C07287=1090.519,65.831,439.779,175.359,18.176,152.786
C07288=1090.524,66.080,439.762,175.361,18.177,152.786
C07289=1090.530,66.329,439.745,175.363,18.179,152.785
C07290=1090.536,66.579,439.729,175.365,18.181,152.785
C07291=1090.541,66.828,439.712,175.367,18.182,152.785
C07292=1090.547,67.078,439.696,175.369,18.183,152.785
C07293=1090.552,67.327,439.679,175.371,18.185,152.785
C07294=1090.559,67.576,439.662,175.373,18.187,152.785
C07295=1090.564,67.826,439.645,175.375,18.188,152.785
C07296=1090.570,68.075,439.629,175.377,18.189,152.785
C07297=1090.575,68.325,439.612,175.379,18.191,152.785
C07298=1090.581,68.574,439.596,175.381,18.192,152.785
C07299=1090.586,68.823,439.578,175.383,18.193,152.785
C07300=1090.592,69.072,439.562,175.385,18.195,152.785
C07301=1090.598,69.322,439.545,175.387,18.197,152.785
C07302=1090.604,69.571,439.528,175.389,18.198,152.785
C07303=1090.609,69.820,439.511,175.391,18.199,152.784
C07304=1090.615,70.070,439.495,175.393,18.201,152.784
C07305=1090.620,70.319,439.478,175.395,18.202,152.784
C07306=1090.627,70.568,439.461,175.397,18.204,152.784
C07307=1090.632,70.818,439.444,175.399,18.205,152.784
C07308=1090.638,71.067,439.428,175.401,18.207,152.784
C07309=1090.643,71.316,439.410,175.403,18.208,152.784
C07310=1090.648,71.566,439.394,175.405,18.210,152.784
C07311=1090.655,71.816,439.377,175.407,18.211,152.784
C07312=1090.660,72.065,439.359,175.409,18.213,152.784
C07313=1090.666,72.314,439.343,175.411,18.214,152.784
C07314=1090.672,72.564,439.326,175.413,18.216,152.784
C07315=1090.677,72.813,439.309,175.415,18.217,152.784
C07316=1090.683,73.062,439.292,175.417,18.218,152.783
C07317=1090.689,73.311,439.275,175.419,18.220,152.783
C07318=1090.694,73.561,439.258,175.421,18.222,152.783
C07319=1090.700,73.810,439.242,175.423,18.223,152.783
C07320=1090.705,74.059,439.224,175.425,18.224,152.783
C07321=1090.711,74.309,439.208,175.427,18.225,152.783
C07322=1090.717,74.559,439.190,175.430,18.227,152.783
C07323=1090.723,74.808,439.173,175.432,18.229,152.783
C07324=1090.729,75.057,439.156,175.433,18.230,152.783
C07325=1090.734,75.307,439.139,175.436,18.232,152.783
C07326=1090.740,75.556,439.122,175.438,18.233,152.783
C07327=1090.746,75.805,439.106,175.440,18.234,152.782
C07328=1090.751,76.054,439.088,175.442,18.236,152.782
C07329=1090.756,76.304,439.071,175.444,18.237,152.782
C07330=1090.762,76.553,439.053,175.446,18.239,152.782
C07331=1090.768,76.803,439.037,175.448,18.240,152.782
C07332=1090.774,77.052,439.019,175.450,18.241,152.782
C07333=1090.779,77.301,439.003,175.452,18.243,152.782
C07334=1090.785,77.550,438.986,175.454,18.244,152.782
C07335=1090.791,77.800,438.969,175.456,18.246,152.782
C07336=1090.797,78.050,438.951,175.458,18.247,152.782
C07337=1090.802,78.299,438.933,175.460,18.248,152.781
C07338=1090.808,78.548,438.917,175.462,18.249,152.781
C07339=1090.814,78.797,438.899,175.464,18.252,152.781
C07340=1090.819,79.047,438.883,175.466,18.253,152.781
C07341=1090.825,79.324,438.863,175.469,18.254,152.781
C07342=1090.832,79.600,438.844,175.471,18.256,152.781
C07343=1090.838,79.877,438.825,175.474,18.257,152.781
C07344=1090.845,80.153,438.805,175.476,18.259,152.781
C07345=1090.850,80.402,438.789,175.478,18.260,152.781
C07346=1090.855,80.651,438.771,175.480,18.262,152.781
C07347=1090.861,80.900,438.753,175.482,18.263,152.781
C07348=1090.867,81.151,438.736,175.484,18.265,152.781
C07349=1090.872,81.400,438.719,175.486,18.266,152.780
C07350=1090.878,81.649,438.701,175.488,18.268,152.780
C07351=1090.883,81.899,438.684,175.491,18.269,152.780
C07352=1090.888,82.148,438.667,175.492,18.270,152.780
C07353=1090.895,82.397,438.649,175.495,18.272,152.780
C07354=1090.901,82.647,438.633,175.496,18.273,152.780
C07355=1090.906,82.896,438.615,175.499,18.275,152.780
C07356=1090.912,83.145,438.597,175.501,18.276,152.780
C07357=1090.917,83.394,438.580,175.503,18.277,152.779
C07358=1090.923,83.644,438.563,175.505,18.278,152.779
C07359=1090.928,83.893,438.545,175.507,18.280,152.779
C07360=1090.934,84.142,438.527,175.510,18.282,152.779
C07361=1090.939,84.391,438.510,175.511,18.283,152.779
C07362=1090.946,84.641,438.492,175.514,18.284,152.779
C07363=1090.951,84.891,438.475,175.516,18.285,152.779
C07364=1090.956,85.140,438.458,175.518,18.287,152.779
C07365=1090.962,85.389,438.440,175.520,18.288,152.779
C07366=1090.968,85.639,438.422,175.522,18.290,152.778
C07367=1090.974,85.888,438.404,175.524,18.291,152.778
C07368=1090.980,86.136,438.388,175.526,18.292,152.778
C07369=1090.986,86.387,438.370,175.529,18.294,152.778
C07370=1090.991,86.636,438.353,175.530,18.295,152.778
C07371=1090.997,86.885,438.335,175.533,18.297,152.778
C07372=1091.002,87.134,438.318,175.535,18.298,152.778
C07373=1091.008,87.384,438.300,175.537,18.299,152.778
C07374=1091.014,87.633,438.282,175.539,18.300,152.778
C07375=1091.019,87.882,438.265,175.541,18.302,152.777
C07376=1091.025,88.131,438.247,175.543,18.303,152.777
C07377=1091.031,88.380,438.229,175.545,18.305,152.777
C07378=1091.036,88.629,438.211,175.548,18.306,152.777
C07379=1091.043,88.879,438.194,175.550,18.307,152.777
C07380=1091.048,89.129,438.177,175.552,18.309,152.777
C07381=1091.053,89.378,438.159,175.554,18.309,152.777
C07382=1091.059,89.628,438.141,175.556,18.311,152.777
C07383=1091.065,89.877,438.124,175.558,18.312,152.776
C07384=1091.070,90.126,438.106,175.561,18.314,152.776
C07385=1091.077,90.375,438.088,175.563,18.315,152.776
C07386=1091.082,90.624,438.071,175.565,18.316,152.776
C07387=1091.087,90.875,438.052,175.567,18.318,152.776
C07388=1091.093,91.124,438.034,175.569,18.319,152.776
C07389=1091.099,91.372,438.016,175.572,18.320,152.776
C07390=1091.105,91.622,437.998,175.573,18.321,152.775
C07391=1091.110,91.871,437.981,175.576,18.323,152.775
C07392=1091.116,92.120,437.963,175.578,18.324,152.775
C07393=1091.121,92.370,437.945,175.580,18.326,152.775
C07394=1091.127,92.619,437.927,175.582,18.327,152.775
C07395=1091.132,92.868,437.909,175.584,18.328,152.775
C07396=1091.139,93.118,437.891,175.587,18.330,152.775
C07397=1091.144,93.367,437.874,175.589,18.331,152.775
C07398=1091.149,93.616,437.856,175.591,18.332,152.774
C07399=1091.155,93.866,437.838,175.593,18.334,152.774
C07400=1091.161,94.114,437.820,175.595,18.335,152.774
C07401=1091.167,94.364,437.802,175.598,18.336,152.774
C07402=1091.172,94.613,437.783,175.599,18.337,152.774
C07403=1091.177,94.862,437.766,175.602,18.339,152.774
C07404=1091.183,95.112,437.748,175.604,18.341,152.774
C07405=1091.189,95.389,437.727,175.607,18.342,152.773
C07406=1091.196,95.666,437.708,175.609,18.343,152.773
C07407=1091.202,95.942,437.688,175.611,18.344,152.773
C07408=1091.208,96.219,437.667,175.614,18.346,152.773
C07409=1091.214,96.468,437.650,175.616,18.347,152.773
C07410=1091.220,96.717,437.632,175.618,18.348,152.773
C07411=1091.225,96.966,437.614,175.621,18.350,152.773
C07412=1091.230,97.215,437.595,175.623,18.351,152.772
C07413=1091.236,97.465,437.577,175.625,18.352,152.772
C07414=1091.242,97.714,437.560,175.627,18.354,152.772
C07415=1091.247,97.964,437.541,175.629,18.355,152.772
C07416=1091.253,98.212,437.523,175.632,18.356,152.772
C07417=1091.259,98.462,437.505,175.634,18.358,152.772
C07418=1091.265,98.711,437.488,175.636,18.358,152.772
C07419=1091.271,98.961,437.468,175.638,18.360,152.771
C07420=1091.276,99.210,437.451,175.640,18.361,152.771
C07421=1091.282,99.459,437.433,175.643,18.362,152.771
C07422=1091.287,99.708,437.414,175.645,18.364,152.771
C07423=1091.293,99.958,437.396,175.647,18.365,152.771
C07424=1091.299,100.207,437.378,175.649,18.367,152.771
C07425=1091.305,100.456,437.359,175.651,18.367,152.770
C07426=1091.310,100.705,437.342,175.654,18.369,152.770
C07427=1091.316,100.955,437.324,175.656,18.370,152.770
C07428=1091.321,101.204,437.305,175.658,18.371,152.770
C07429=1091.327,101.454,437.287,175.661,18.373,152.770
C07430=1091.333,101.702,437.268,175.662,18.374,152.770
C07431=1091.339,101.952,437.250,175.665,18.375,152.769
C07432=1091.343,102.201,437.232,175.668,18.376,152.769
C07433=1091.350,102.451,437.213,175.669,18.377,152.769
C07434=1091.355,102.700,437.195,175.672,18.379,152.769
C07435=1091.361,102.949,437.176,175.675,18.380,152.769
C07436=1091.366,103.198,437.158,175.676,18.381,152.769
C07437=1091.372,103.448,437.140,175.679,18.383,152.769
C07438=1091.377,103.697,437.121,175.681,18.383,152.768
C07439=1091.383,103.946,437.103,175.683,18.385,152.768
C07440=1091.388,104.195,437.085,175.686,18.387,152.768
C07441=1091.395,104.444,437.066,175.688,18.387,152.768
C07442=1091.399,104.694,437.048,175.690,18.389,152.768
C07443=1091.406,104.943,437.029,175.693,18.390,152.768
C07444=1091.411,105.192,437.011,175.694,18.391,152.767
C07445=1091.417,105.441,436.992,175.697,18.393,152.767
C07446=1091.422,105.691,436.974,175.699,18.393,152.767
C07447=1091.428,105.940,436.956,175.701,18.395,152.767
C07448=1091.433,106.189,436.937,175.704,18.396,152.767
C07449=1091.439,106.439,436.918,175.706,18.397,152.767
C07450=1091.445,106.688,436.900,175.708,18.399,152.766
C07451=1091.450,106.937,436.881,175.711,18.400,152.766
C07452=1091.456,107.186,436.863,175.713,18.401,152.766
C07453=1091.461,107.435,436.844,175.715,18.402,152.766
C07454=1091.468,107.685,436.826,175.718,18.404,152.766
C07455=1091.473,107.934,436.807,175.720,18.405,152.766
C07456=1091.478,108.183,436.788,175.722,18.406,152.765
C07457=1091.484,108.433,436.770,175.724,18.407,152.765
C07458=1091.490,108.681,436.751,175.727,18.408,152.765
C07459=1091.496,108.931,436.732,175.729,18.410,152.765
C07460=1091.501,109.181,436.714,175.731,18.410,152.765
C07461=1091.506,109.429,436.695,175.734,18.412,152.764
C07462=1091.513,109.678,436.676,175.736,18.413,152.764
C07463=1091.518,109.928,436.658,175.738,18.414,152.764
C07464=1091.524,110.177,436.639,175.741,18.415,152.764
C07465=1091.530,110.426,436.620,175.743,18.417,152.764
C07466=1091.535,110.675,436.601,175.745,18.417,152.763
C07467=1091.541,110.925,436.583,175.748,18.419,152.763
C07468=1091.547,111.174,436.564,175.750,18.420,152.763
C07469=1091.553,111.451,436.544,175.752,18.421,152.763
C07470=1091.560,111.727,436.522,175.755,18.422,152.763
C07471=1091.566,112.004,436.502,175.757,18.424,152.763
C07472=1091.572,112.281,436.481,175.760,18.425,152.762
C07473=1091.578,112.530,436.462,175.763,18.426,152.762
C07474=1091.583,112.779,436.443,175.765,18.428,152.762
C07475=1091.588,113.029,436.425,175.767,18.428,152.762
C07476=1091.595,113.278,436.406,175.770,18.430,152.762
C07477=1091.600,113.527,436.387,175.772,18.431,152.761
C07478=1091.605,113.776,436.368,175.774,18.432,152.761
C07479=1091.611,114.025,436.349,175.777,18.433,152.761
C07480=1091.617,114.275,436.330,175.779,18.435,152.761
C07481=1091.623,114.523,436.311,175.781,18.435,152.761
C07482=1091.628,114.773,436.292,175.784,18.437,152.760
C07483=1091.634,115.023,436.273,175.786,18.438,152.760
C07484=1091.639,115.272,436.254,175.788,18.439,152.760
C07485=1091.644,115.521,436.235,175.791,18.440,152.760
C07486=1091.650,115.770,436.216,175.793,18.442,152.760
C07487=1091.655,116.019,436.197,175.795,18.442,152.759
C07488=1091.661,116.269,436.178,175.798,18.444,152.759
C07489=1091.667,116.518,436.158,175.801,18.445,152.759
C07490=1091.672,116.767,436.140,175.802,18.446,152.759
C07491=1091.677,117.016,436.120,175.805,18.447,152.759
C07492=1091.684,117.265,436.102,175.808,18.448,152.758
C07493=1091.689,117.514,436.083,175.809,18.450,152.758
C07494=1091.694,117.763,436.064,175.812,18.451,152.758
C07495=1091.700,118.013,436.044,175.815,18.452,152.758
C07496=1091.705,118.262,436.025,175.816,18.453,152.758
C07497=1091.711,118.511,436.006,175.819,18.454,152.757
C07498=1091.717,118.760,435.987,175.822,18.456,152.757
C07499=1091.722,119.010,435.968,175.824,18.456,152.757
C07500=1091.727,119.259,435.949,175.826,18.458,152.757
C07501=1091.733,119.508,435.930,175.829,18.459,152.757
C07502=1091.739,119.758,435.910,175.832,18.460,152.756
C07503=1091.744,120.007,435.891,175.833,18.461,152.756
C07504=1091.750,120.256,435.872,175.836,18.462,152.756
C07505=1091.756,120.504,435.852,175.839,18.463,152.756
C07506=1091.761,120.754,435.833,175.840,18.464,152.756
C07507=1091.767,121.003,435.814,175.843,18.465,152.755
C07508=1091.772,121.252,435.795,175.846,18.467,152.755
C07509=1091.778,121.502,435.776,175.848,18.468,152.755
C07510=1091.783,121.751,435.756,175.850,18.469,152.755
C07511=1091.789,122.000,435.737,175.853,18.470,152.755
C07512=1091.795,122.249,435.717,175.855,18.471,152.754
C07513=1091.800,122.498,435.698,175.858,18.472,152.754
C07514=1091.806,122.747,435.679,175.860,18.473,152.754
C07515=1091.812,122.997,435.660,175.863,18.474,152.754
C07516=1091.817,123.246,435.641,175.865,18.475,152.754
C07517=1091.823,123.495,435.621,175.867,18.477,152.753
C07518=1091.828,123.744,435.601,175.870,18.478,152.753
C07519=1091.833,123.994,435.582,175.872,18.478,152.753
C07520=1091.839,124.243,435.563,175.875,18.480,152.753
C07521=1091.845,124.492,435.543,175.877,18.481,152.752
C07522=1091.851,124.741,435.524,175.879,18.482,152.752
C07523=1091.856,124.991,435.504,175.882,18.483,152.752
C07524=1091.862,125.239,435.484,175.885,18.484,152.752
C07525=1091.867,125.488,435.465,175.887,18.485,152.751
C07526=1091.873,125.738,435.446,175.889,18.486,152.751
C07527=1091.879,125.986,435.426,175.892,18.487,152.751
C07528=1091.885,126.236,435.407,175.895,18.488,152.751
C07529=1091.890,126.485,435.388,175.897,18.489,152.750
C07530=1091.896,126.734,435.367,175.899,18.490,152.750
C07531=1091.901,126.984,435.348,175.902,18.492,152.750
C07532=1091.907,127.233,435.329,175.904,18.492,152.750
C07533=1091.913,127.509,435.308,175.907,18.494,152.750
C07534=1091.920,127.786,435.285,175.910,18.495,152.749
C07535=1091.926,128.063,435.263,175.913,18.496,152.749
C07536=1091.932,128.339,435.242,175.916,18.497,152.749
C07537=1091.938,128.588,435.223,175.917,18.498,152.749
C07538=1091.943,128.838,435.202,175.920,18.499,152.748
C07539=1091.949,129.087,435.183,175.923,18.500,152.748
C07540=1091.955,129.336,435.163,175.925,18.501,152.748
C07541=1091.961,129.585,435.144,175.928,18.502,152.747
C07542=1091.967,129.834,435.124,175.930,18.503,152.747
C07543=1091.972,130.084,435.105,175.933,18.504,152.747
C07544=1091.978,130.332,435.085,175.935,18.505,152.747
C07545=1091.983,130.582,435.065,175.938,18.506,152.746
C07546=1091.989,130.831,435.045,175.940,18.507,152.746
C07547=1091.995,131.080,435.026,175.942,18.508,152.746
C07548=1092.001,131.329,435.006,175.945,18.509,152.746
C07549=1092.007,131.579,434.986,175.948,18.510,152.746
C07550=1092.012,131.828,434.966,175.950,18.511,152.745
C07551=1092.018,132.077,434.947,175.952,18.512,152.745
C07552=1092.024,132.326,434.927,175.955,18.513,152.745
C07553=1092.029,132.575,434.907,175.958,18.514,152.744
C07554=1092.035,132.824,434.887,175.961,18.515,152.744
C07555=1092.041,133.073,434.867,175.962,18.516,152.744
C07556=1092.046,133.323,434.848,175.965,18.517,152.744
C07557=1092.052,133.572,434.827,175.968,18.518,152.743
C07558=1092.057,133.821,434.808,175.971,18.519,152.743
C07559=1092.062,134.070,434.787,175.973,18.520,152.743
C07560=1092.068,134.319,434.767,175.975,18.521,152.743
C07561=1092.074,134.569,434.748,175.978,18.522,152.742
C07562=1092.079,134.818,434.727,175.981,18.523,152.742
C07563=1092.085,135.067,434.708,175.983,18.524,152.742
C07564=1092.090,135.316,434.688,175.986,18.525,152.742
C07565=1092.096,135.565,434.668,175.988,18.526,152.741
C07566=1092.102,135.814,434.648,175.991,18.527,152.741
C07567=1092.108,136.063,434.627,175.993,18.528,152.741
C07568=1092.113,136.313,434.608,175.996,18.529,152.741
C07569=1092.119,136.562,434.587,175.998,18.530,152.740
C07570=1092.125,136.810,434.567,176.001,18.531,152.740
C07571=1092.131,137.059,434.547,176.003,18.532,152.740
C07572=1092.135,137.309,434.528,176.006,18.533,152.740
C07573=1092.141,137.558,434.508,176.009,18.534,152.739
C07574=1092.147,137.807,434.487,176.011,18.535,152.739
C07575=1092.153,138.056,434.467,176.013,18.536,152.739
C07576=1092.158,138.306,434.447,176.016,18.537,152.739
C07577=1092.164,138.554,434.427,176.019,18.538,152.738
C07578=1092.169,138.803,434.407,176.021,18.539,152.738
C07579=1092.175,139.052,434.387,176.024,18.539,152.738
C07580=1092.180,139.301,434.366,176.026,18.540,152.737
C07581=1092.187,139.551,434.346,176.029,18.541,152.737
C07582=1092.192,139.801,434.326,176.032,18.543,152.737
C07583=1092.198,140.049,434.306,176.034,18.543,152.737
C07584=1092.203,140.299,434.286,176.037,18.544,152.736
C07585=1092.209,140.547,434.266,176.039,18.545,152.736
C07586=1092.214,140.797,434.245,176.042,18.547,152.736
C07587=1092.219,141.046,434.225,176.045,18.548,152.736
C07588=1092.225,141.294,434.205,176.047,18.548,152.735
C07589=1092.231,141.544,434.184,176.050,18.549,152.735
C07590=1092.237,141.792,434.164,176.052,18.550,152.735
C07591=1092.242,142.042,434.144,176.055,18.551,152.734
C07592=1092.248,142.291,434.123,176.057,18.552,152.734
C07593=1092.254,142.540,434.103,176.060,18.553,152.734
C07594=1092.259,142.789,434.082,176.063,18.554,152.734
C07595=1092.264,143.038,434.062,176.065,18.555,152.733
C07596=1092.270,143.287,434.042,176.068,18.556,152.733
C07597=1092.276,143.564,434.019,176.071,18.557,152.733
C07598=1092.282,143.841,433.996,176.074,18.558,152.732
C07599=1092.289,144.118,433.974,176.077,18.559,152.732
C07600=1092.295,144.394,433.951,176.080,18.560,152.732
C07601=1092.301,144.643,433.930,176.082,18.561,152.731
C07602=1092.306,144.892,433.910,176.085,18.562,152.731
C07603=1092.312,145.141,433.890,176.087,18.563,152.731
C07604=1092.317,145.390,433.869,176.090,18.564,152.731
C07605=1092.322,145.639,433.849,176.093,18.564,152.730
C07606=1092.329,145.889,433.828,176.095,18.566,152.730
C07607=1092.334,146.137,433.807,176.097,18.566,152.730
C07608=1092.340,146.387,433.787,176.100,18.567,152.730
C07609=1092.346,146.635,433.767,176.103,18.568,152.729
C07610=1092.351,146.884,433.746,176.106,18.569,152.729
C07611=1092.357,147.134,433.725,176.109,18.570,152.729
C07612=1092.362,147.383,433.705,176.111,18.571,152.728
C07613=1092.368,147.632,433.684,176.114,18.571,152.728
C07614=1092.374,147.881,433.663,176.116,18.573,152.728
C07615=1092.379,148.130,433.643,176.119,18.574,152.727
C07616=1092.385,148.380,433.622,176.122,18.574,152.727
C07617=1092.391,148.628,433.602,176.125,18.575,152.727
C07618=1092.396,148.877,433.581,176.127,18.576,152.727
C07619=1092.402,149.126,433.560,176.129,18.577,152.726
C07620=1092.407,149.376,433.539,176.132,18.578,152.726
C07621=1092.413,149.625,433.519,176.135,18.579,152.726
C07622=1092.418,149.874,433.497,176.138,18.580,152.725
C07623=1092.424,150.122,433.477,176.140,18.581,152.725
C07624=1092.430,150.372,433.457,176.143,18.581,152.725
C07625=1092.435,150.621,433.436,176.146,18.582,152.724
C07626=1092.441,150.870,433.415,176.148,18.584,152.724
C07627=1092.446,151.119,433.394,176.151,18.584,152.724
C07628=1092.452,151.369,433.373,176.153,18.585,152.724
C07629=1092.458,151.617,433.352,176.156,18.586,152.723
C07630=1092.463,151.866,433.331,176.159,18.587,152.723
C07631=1092.468,152.116,433.311,176.162,18.588,152.723
C07632=1092.474,152.365,433.289,176.164,18.589,152.722
C07633=1092.479,152.614,433.269,176.167,18.590,152.722
C07634=1092.486,152.862,433.248,176.169,18.590,152.722
C07635=1092.491,153.111,433.227,176.172,18.591,152.721
C07636=1092.497,153.361,433.206,176.175,18.592,152.721
C07637=1092.502,153.610,433.185,176.178,18.593,152.721
C07638=1092.508,153.859,433.165,176.181,18.594,152.720
C07639=1092.514,154.108,433.143,176.184,18.595,152.720
C07640=1092.519,154.357,433.122,176.186,18.595,152.720
C07641=1092.525,154.605,433.101,176.189,18.596,152.719
C07642=1092.531,154.855,433.080,176.191,18.597,152.719
C07643=1092.536,155.104,433.059,176.194,18.598,152.719
C07644=1092.541,155.353,433.038,176.197,18.599,152.719
C07645=1092.548,155.602,433.017,176.200,18.600,152.718
C07646=1092.553,155.851,432.996,176.202,18.600,152.718
C07647=1092.558,156.100,432.975,176.205,18.601,152.718
C07648=1092.564,156.350,432.954,176.208,18.602,152.717
C07649=1092.570,156.598,432.933,176.210,18.603,152.717
C07650=1092.575,156.847,432.912,176.213,18.604,152.717
C07651=1092.581,157.096,432.891,176.216,18.605,152.716
C07652=1092.586,157.346,432.869,176.219,18.606,152.716
C07653=1092.591,157.594,432.848,176.221,18.606,152.716
C07654=1092.597,157.844,432.827,176.224,18.607,152.715
C07655=1092.603,158.093,432.806,176.227,18.608,152.715
C07656=1092.608,158.341,432.785,176.230,18.609,152.715
C07657=1092.614,158.591,432.764,176.233,18.610,152.714
C07658=1092.620,158.840,432.743,176.235,18.611,152.714
C07659=1092.626,159.089,432.721,176.237,18.612,152.714
C07660=1092.631,159.338,432.700,176.240,18.612,152.713
C07661=1092.637,159.614,432.676,176.244,18.613,152.713
C07662=1092.643,159.891,432.653,176.247,18.615,152.713
C07663=1092.650,160.167,432.630,176.250,18.615,152.712
C07664=1092.656,160.443,432.606,176.253,18.616,152.712
C07665=1092.662,160.692,432.584,176.256,18.617,152.712
C07666=1092.667,160.941,432.563,176.259,18.618,152.711
C07667=1092.673,161.191,432.541,176.261,18.619,152.711
C07668=1092.678,161.439,432.520,176.263,18.619,152.711
C07669=1092.684,161.688,432.499,176.266,18.620,152.710
C07670=1092.690,161.938,432.478,176.269,18.621,152.710
C07671=1092.694,162.186,432.456,176.272,18.622,152.710
C07672=1092.700,162.435,432.435,176.275,18.622,152.709
C07673=1092.706,162.684,432.413,176.278,18.624,152.709
C07674=1092.711,162.933,432.392,176.281,18.624,152.709
C07675=1092.717,163.183,432.370,176.283,18.625,152.708
C07676=1092.722,163.432,432.348,176.286,18.627,152.708
C07677=1092.727,163.680,432.327,176.288,18.627,152.708
C07678=1092.733,163.929,432.305,176.291,18.628,152.707
C07679=1092.738,164.178,432.284,176.294,18.628,152.707
C07680=1092.744,164.428,432.263,176.297,18.630,152.707
C07681=1092.749,164.677,432.241,176.300,18.630,152.706
C07682=1092.754,164.925,432.220,176.303,18.631,152.706
C07683=1092.760,165.175,432.197,176.306,18.632,152.706
C07684=1092.765,165.423,432.176,176.308,18.633,152.705
C07685=1092.772,165.672,432.154,176.311,18.634,152.705
C07686=1092.776,165.921,432.133,176.313,18.634,152.705
C07687=1092.783,166.170,432.111,176.316,18.635,152.704
C07688=1092.787,166.419,432.089,176.319,18.636,152.704
C07689=1092.794,166.668,432.067,176.322,18.637,152.704
C07690=1092.798,166.917,432.046,176.325,18.638,152.703
C07691=1092.804,167.166,432.024,176.328,18.639,152.703
C07692=1092.809,167.415,432.002,176.331,18.639,152.703
C07693=1092.815,167.664,431.981,176.333,18.641,152.702
C07694=1092.820,167.913,431.959,176.336,18.641,152.702
C07695=1092.826,168.162,431.937,176.339,18.642,152.702
C07696=1092.831,168.411,431.915,176.341,18.642,152.701
C07697=1092.837,168.660,431.894,176.344,18.643,152.701
C07698=1092.842,168.909,431.872,176.347,18.644,152.701
C07699=1092.848,169.158,431.850,176.350,18.645,152.700
C07700=1092.853,169.407,431.828,176.353,18.646,152.700
C07701=1092.859,169.657,431.806,176.356,18.647,152.700
C07702=1092.864,169.905,431.785,176.359,18.647,152.699
C07703=1092.870,170.155,431.763,176.362,18.648,152.699
C07704=1092.875,170.403,431.741,176.365,18.649,152.699
C07705=1092.881,170.653,431.719,176.368,18.650,152.698
C07706=1092.887,170.901,431.697,176.371,18.651,152.698
C07707=1092.893,171.150,431.675,176.373,18.652,152.697
C07708=1092.898,171.399,431.653,176.375,18.652,152.697
C07709=1092.904,171.648,431.632,176.378,18.652,152.697
C07710=1092.909,171.898,431.609,176.381,18.654,152.696
C07711=1092.915,172.146,431.588,176.384,18.654,152.696
C07712=1092.920,172.395,431.565,176.387,18.655,152.696
C07713=1092.926,172.643,431.544,176.390,18.656,152.695
C07714=1092.931,172.893,431.522,176.393,18.657,152.695
C07715=1092.937,173.142,431.500,176.396,18.657,152.695
C07716=1092.943,173.390,431.478,176.399,18.658,152.694
C07717=1092.948,173.640,431.455,176.402,18.659,152.694
C07718=1092.954,173.888,431.434,176.405,18.660,152.693
C07719=1092.959,174.138,431.412,176.408,18.661,152.693
C07720=1092.965,174.387,431.389,176.411,18.661,152.693
C07721=1092.970,174.635,431.368,176.413,18.662,152.692
C07722=1092.976,174.885,431.345,176.416,18.662,152.692
C07723=1092.982,175.133,431.323,176.419,18.663,152.692
C07724=1092.987,175.382,431.301,176.422,18.664,152.691
C07725=1092.994,175.659,431.277,176.425,18.665,152.691
C07726=1093.000,175.934,431.252,176.428,18.666,152.690
C07727=1093.006,176.210,431.227,176.431,18.666,152.690
C07728=1093.013,176.486,431.203,176.434,18.667,152.690
C07729=1093.018,176.735,431.180,176.437,18.668,152.689
C07730=1093.023,176.984,431.158,176.440,18.668,152.689
C07731=1093.029,177.233,431.137,176.443,18.669,152.689
C07732=1093.035,177.482,431.114,176.446,18.670,152.688
C07733=1093.040,177.732,431.092,176.449,18.671,152.688
C07734=1093.046,177.980,431.070,176.452,18.671,152.687
C07735=1093.052,178.229,431.047,176.455,18.672,152.687
C07736=1093.057,178.478,431.025,176.458,18.673,152.687
C07737=1093.064,178.727,431.003,176.461,18.673,152.686
C07738=1093.069,178.975,430.980,176.464,18.674,152.686
C07739=1093.074,179.225,430.958,176.467,18.675,152.685
C07740=1093.081,179.473,430.936,176.470,18.676,152.685
C07741=1093.086,179.723,430.913,176.473,18.677,152.685
C07742=1093.091,179.971,430.891,176.476,18.677,152.684
C07743=1093.097,180.220,430.869,176.479,18.678,152.684
C07744=1093.103,180.469,430.846,176.482,18.679,152.683
C07745=1093.109,180.719,430.824,176.485,18.679,152.683
C07746=1093.114,180.968,430.801,176.488,18.680,152.683
C07747=1093.120,181.216,430.779,176.490,18.680,152.682
C07748=1093.126,181.465,430.757,176.493,18.681,152.682
C07749=1093.131,181.714,430.734,176.496,18.681,152.681
C07750=1093.137,181.964,430.712,176.499,18.682,152.681
C07751=1093.143,182.212,430.689,176.502,18.683,152.681
C07752=1093.149,182.461,430.666,176.505,18.683,152.680
C07753=1093.154,182.710,430.645,176.508,18.684,152.680
C07754=1093.159,182.959,430.622,176.511,18.685,152.679
C07755=1093.166,183.207,430.599,176.514,18.685,152.679
C07756=1093.171,183.457,430.577,176.517,18.686,152.679
C07757=1093.177,183.706,430.554,176.520,18.687,152.678
C07758=1093.183,183.955,430.531,176.523,18.688,152.678
C07759=1093.189,184.203,430.509,176.526,18.688,152.677
C07760=1093.194,184.452,430.487,176.529,18.689,152.677
C07761=1093.200,184.701,430.464,176.532,18.690,152.677
C07762=1093.206,184.950,430.441,176.535,18.690,152.676
C07763=1093.211,185.199,430.418,176.538,18.691,152.676
C07764=1093.217,185.448,430.396,176.541,18.692,152.675
C07765=1093.222,185.697,430.373,176.544,18.692,152.675
C07766=1093.228,185.945,430.350,176.547,18.693,152.675
C07767=1093.233,186.194,430.327,176.550,18.694,152.674
C07768=1093.239,186.443,430.304,176.553,18.694,152.674
C07769=1093.244,186.693,430.282,176.556,18.695,152.673
C07770=1093.250,186.942,430.259,176.559,18.696,152.673
C07771=1093.255,187.190,430.237,176.562,18.697,152.673
C07772=1093.261,187.439,430.214,176.565,18.697,152.672
C07773=1093.266,187.688,430.190,176.568,18.698,152.672
C07774=1093.272,187.937,430.167,176.571,18.699,152.672
C07775=1093.277,188.186,430.145,176.574,18.699,152.671
C07776=1093.283,188.435,430.122,176.577,18.700,152.671
C07777=1093.288,188.683,430.100,176.580,18.701,152.670
C07778=1093.294,188.932,430.077,176.583,18.701,152.670
C07779=1093.300,189.181,430.054,176.586,18.702,152.670
C07780=1093.305,189.430,430.030,176.589,18.703,152.669
C07781=1093.310,189.679,430.007,176.592,18.704,152.669
C07782=1093.316,189.928,429.984,176.595,18.704,152.668
C07783=1093.322,190.177,429.961,176.598,18.705,152.668
C07784=1093.327,190.425,429.939,176.601,18.706,152.668
C07785=1093.333,190.674,429.916,176.604,18.706,152.667
C07786=1093.338,190.923,429.892,176.607,18.707,152.667
C07787=1093.343,191.172,429.869,176.610,18.708,152.666
C07788=1093.349,191.421,429.846,176.613,18.709,152.666
C07789=1093.355,191.697,429.821,176.616,18.709,152.666
C07790=1093.361,191.972,429.796,176.619,18.710,152.665
C07791=1093.368,192.248,429.769,176.623,18.711,152.665
C07792=1093.374,192.524,429.744,176.626,18.712,152.664
C07793=1093.379,192.773,429.721,176.629,18.712,152.664
C07794=1093.385,193.021,429.698,176.632,18.713,152.663
C07795=1093.391,193.270,429.675,176.635,18.714,152.663
C07796=1093.396,193.520,429.651,176.638,18.714,152.663
C07797=1093.402,193.768,429.628,176.641,18.715,152.662
C07798=1093.407,194.017,429.605,176.644,18.716,152.662
C07799=1093.413,194.266,429.582,176.647,18.716,152.661
C07800=1093.418,194.515,429.558,176.650,18.717,152.661
C07801=1093.424,194.764,429.535,176.653,18.718,152.661
C07802=1093.430,195.013,429.512,176.656,18.718,152.660
C07803=1093.436,195.261,429.489,176.660,18.719,152.660
C07804=1093.441,195.510,429.465,176.663,18.719,152.659
C07805=1093.446,195.759,429.442,176.666,18.721,152.659
C07806=1093.452,196.008,429.419,176.669,18.721,152.658
C07807=1093.458,196.256,429.396,176.672,18.722,152.658
C07808=1093.463,196.505,429.372,176.675,18.723,152.658
C07809=1093.469,196.754,429.349,176.678,18.723,152.657
C07810=1093.475,197.003,429.326,176.681,18.724,152.657
C07811=1093.480,197.252,429.302,176.685,18.724,152.656
C07812=1093.486,197.501,429.279,176.688,18.725,152.656
C07813=1093.491,197.750,429.256,176.691,18.726,152.655
C07814=1093.497,197.998,429.232,176.694,18.726,152.655
C07815=1093.502,198.247,429.209,176.697,18.727,152.655
C07816=1093.508,198.496,429.186,176.700,18.728,152.654
C07817=1093.514,198.744,429.162,176.703,18.728,152.654
C07818=1093.519,198.993,429.139,176.706,18.728,152.653
C07819=1093.526,199.242,429.115,176.709,18.729,152.653
C07820=1093.531,199.492,429.091,176.713,18.730,152.653
C07821=1093.537,199.741,429.068,176.716,18.731,152.652
C07822=1093.543,199.989,429.045,176.719,18.731,152.652
C07823=1093.548,200.238,429.021,176.722,18.732,152.651
C07824=1093.554,200.486,428.997,176.725,18.733,152.651
C07825=1093.559,200.735,428.974,176.728,18.733,152.650
C07826=1093.565,200.984,428.950,176.731,18.734,152.650
C07827=1093.571,201.233,428.927,176.734,18.734,152.649
C07828=1093.577,201.482,428.903,176.737,18.735,152.649
C07829=1093.582,201.731,428.880,176.740,18.736,152.649
C07830=1093.588,201.979,428.856,176.743,18.736,152.648
C07831=1093.593,202.228,428.832,176.746,18.737,152.648
C07832=1093.599,202.477,428.809,176.749,18.737,152.647
C07833=1093.605,202.726,428.786,176.753,18.738,152.647
C07834=1093.611,202.975,428.761,176.756,18.739,152.646
C07835=1093.616,203.224,428.738,176.759,18.739,152.646
C07836=1093.622,203.472,428.714,176.762,18.740,152.646
C07837=1093.627,203.721,428.690,176.765,18.741,152.645
C07838=1093.633,203.970,428.667,176.768,18.741,152.645
C07839=1093.638,204.218,428.643,176.772,18.742,152.644
C07840=1093.644,204.468,428.619,176.775,18.742,152.644
C07841=1093.650,204.717,428.595,176.778,18.743,152.643
C07842=1093.655,204.965,428.571,176.781,18.744,152.643
C07843=1093.661,205.214,428.548,176.784,18.745,152.643
C07844=1093.666,205.463,428.524,176.788,18.745,152.642
C07845=1093.671,205.711,428.499,176.791,18.746,152.642
C07846=1093.678,205.961,428.476,176.794,18.747,152.641
C07847=1093.683,206.209,428.452,176.797,18.747,152.641
C07848=1093.689,206.458,428.428,176.800,18.748,152.641
C07849=1093.694,206.706,428.404,176.803,18.748,152.640
C07850=1093.699,206.955,428.380,176.806,18.749,152.640
C07851=1093.706,207.204,428.356,176.810,18.750,152.639
C07852=1093.711,207.453,428.332,176.813,18.751,152.639
C07853=1093.734,208.471,428.234,176.870,18.776,152.634
C07854=1093.742,208.846,428.197,176.874,18.778,152.634
C07855=1093.751,209.221,428.161,176.878,18.781,152.633
C07856=1093.759,209.597,428.124,176.884,18.784,152.633
C07857=1093.768,209.972,428.087,176.888,18.785,152.633
C07858=1093.773,210.221,428.063,176.891,18.787,152.632
C07859=1093.779,210.470,428.038,176.894,18.789,152.632
C07860=1093.785,210.719,428.014,176.897,18.790,152.632
C07861=1093.791,210.968,427.989,176.899,18.791,152.632
C07862=1093.796,211.217,427.965,176.903,18.793,152.632
C07863=1093.801,211.465,427.941,176.906,18.794,152.631
C07864=1093.807,211.714,427.916,176.909,18.796,152.631
C07865=1093.813,211.962,427.891,176.912,18.798,152.631
C07866=1093.818,212.211,427.867,176.915,18.799,152.631
C07867=1093.824,212.460,427.842,176.918,18.801,152.630
C07868=1093.829,212.709,427.818,176.921,18.802,152.630
C07869=1093.835,212.958,427.793,176.924,18.804,152.630
C07870=1093.841,213.206,427.768,176.927,18.805,152.630
C07871=1093.847,213.455,427.744,176.930,18.807,152.630
C07872=1093.852,213.704,427.720,176.933,18.808,152.629
C07873=1093.857,213.953,427.695,176.936,18.810,152.629
C07874=1093.863,214.202,427.671,176.939,18.811,152.629
C07875=1093.869,214.450,427.646,176.942,18.813,152.629
C07876=1093.875,214.699,427.621,176.945,18.815,152.629
C07877=1093.880,214.948,427.597,176.948,18.816,152.628
C07878=1093.886,215.196,427.572,176.951,18.818,152.628
C07879=1093.891,215.445,427.547,176.954,18.819,152.628
C07880=1093.897,215.694,427.523,176.958,18.821,152.628
C07881=1093.902,215.943,427.497,176.960,18.823,152.628
C07882=1093.907,216.191,427.473,176.964,18.824,152.627
C07883=1093.913,216.440,427.448,176.966,18.825,152.627
C07884=1093.919,216.688,427.423,176.969,18.827,152.627
C07885=1093.925,216.938,427.399,176.972,18.829,152.627
C07886=1093.930,217.186,427.374,176.975,18.830,152.627
C07887=1093.936,217.435,427.348,176.978,18.832,152.626
C07888=1093.941,217.684,427.324,176.981,18.833,152.626
C07889=1093.947,217.933,427.299,176.985,18.835,152.626
C07890=1093.952,218.181,427.275,176.987,18.837,152.626
C07891=1093.959,218.430,427.249,176.991,18.838,152.626
C07892=1093.964,218.678,427.225,176.994,18.840,152.625
C07893=1093.969,218.927,427.199,176.997,18.841,152.625
C07894=1093.975,219.176,427.175,177.000,18.843,152.625
C07895=1093.981,219.425,427.149,177.003,18.845,152.625
C07896=1093.986,219.673,427.125,177.006,18.846,152.624
C07897=1093.992,219.922,427.100,177.009,18.848,152.624
C07898=1093.997,220.170,427.074,177.012,18.849,152.624
C07899=1094.003,220.419,427.050,177.015,18.850,152.624
C07900=1094.009,220.667,427.025,177.018,18.852,152.624
C07901=1094.015,220.917,427.000,177.021,18.854,152.623
C07902=1094.020,221.166,426.974,177.024,18.855,152.623
C07903=1094.026,221.414,426.949,177.027,18.857,152.623
C07904=1094.032,221.663,426.925,177.030,18.859,152.623
C07905=1094.037,221.911,426.900,177.033,18.860,152.623
C07906=1094.046,222.291,426.861,177.038,18.863,152.622
C07907=1094.054,222.670,426.822,177.043,18.865,152.622
C07908=1094.063,223.049,426.784,177.047,18.867,152.622
C07909=1094.072,223.430,426.745,177.052,18.870,152.621
C07910=1094.077,223.678,426.720,177.055,18.871,152.621
C07911=1094.082,223.927,426.695,177.058,18.873,152.621
C07912=1094.088,224.175,426.670,177.061,18.875,152.621
C07913=1094.093,224.424,426.644,177.064,18.877,152.621
C07914=1094.100,224.673,426.619,177.067,18.878,152.620
C07915=1094.104,224.922,426.594,177.071,18.880,152.620
C07916=1094.110,225.170,426.569,177.073,18.881,152.620
C07917=1094.117,225.419,426.543,177.077,18.883,152.620
C07918=1094.121,225.667,426.518,177.079,18.884,152.620
C07919=1094.128,225.916,426.492,177.083,18.886,152.619
C07920=1094.132,226.164,426.467,177.085,18.888,152.619
C07921=1094.138,226.413,426.442,177.089,18.889,152.619
C07922=1094.144,226.662,426.416,177.092,18.891,152.619
C07923=1094.150,226.911,426.391,177.095,18.893,152.619
C07924=1094.155,227.159,426.365,177.098,18.894,152.618
C07925=1094.161,227.408,426.340,177.101,18.896,152.618
C07926=1094.167,227.657,426.314,177.104,18.897,152.618
C07927=1094.172,227.905,426.289,177.107,18.899,152.618
C07928=1094.178,228.154,426.263,177.110,18.901,152.618
C07929=1094.184,228.403,426.238,177.113,18.902,152.617
C07930=1094.189,228.651,426.212,177.116,18.903,152.617
C07931=1094.195,228.900,426.187,177.120,18.906,152.617
C07932=1094.200,229.149,426.161,177.123,18.907,152.617
C07933=1094.207,229.397,426.136,177.126,18.909,152.617
C07934=1094.211,229.646,426.110,177.129,18.911,152.616
C07935=1094.217,229.895,426.084,177.132,18.912,152.616
C07936=1094.223,230.143,426.059,177.135,18.914,152.616
C07937=1094.229,230.392,426.033,177.138,18.915,152.616
C07938=1094.235,230.641,426.008,177.141,18.917,152.616
C07939=1094.240,230.889,425.982,177.144,18.919,152.615
C07940=1094.245,231.138,425.956,177.147,18.920,152.615
C07941=1094.252,231.386,425.930,177.150,18.922,152.615
C07942=1094.257,231.635,425.904,177.154,18.924,152.615
C07943=1094.262,231.883,425.879,177.157,18.925,152.615
C07944=1094.268,232.132,425.853,177.160,18.927,152.614
C07945=1094.274,232.381,425.827,177.163,18.929,152.614
C07946=1094.279,232.630,425.801,177.166,18.930,152.614
C07947=1094.284,232.878,425.775,177.169,18.932,152.614
C07948=1094.291,233.126,425.750,177.172,18.933,152.614
C07949=1094.296,233.375,425.724,177.175,18.936,152.614
C07950=1094.301,233.624,425.698,177.178,18.937,152.613
C07951=1094.307,233.873,425.671,177.182,18.938,152.613
C07952=1094.313,234.121,425.646,177.185,18.941,152.613
C07953=1094.318,234.370,425.620,177.188,18.942,152.613
C07954=1094.324,234.619,425.594,177.191,18.944,152.613
C07955=1094.330,234.867,425.568,177.194,18.945,152.612
C07956=1094.335,235.116,425.542,177.197,18.947,152.612
C07957=1094.340,235.364,425.516,177.200,18.948,152.612
C07958=1094.349,235.735,425.477,177.205,18.951,152.612
C07959=1094.357,236.106,425.438,177.209,18.954,152.611
C07960=1094.365,236.477,425.400,177.213,18.956,152.611
C07961=1094.374,236.848,425.361,177.219,18.959,152.611
C07962=1094.379,237.097,425.335,177.221,18.960,152.611
C07963=1094.385,237.345,425.308,177.225,18.963,152.611
C07964=1094.391,237.594,425.283,177.228,18.964,152.610
C07965=1094.397,237.842,425.256,177.231,18.965,152.610
C07966=1094.402,238.091,425.230,177.234,18.968,152.610
C07967=1094.408,238.339,425.203,177.237,18.969,152.610
C07968=1094.414,238.588,425.177,177.240,18.971,152.610
C07969=1094.419,238.837,425.151,177.244,18.973,152.609
C07970=1094.424,239.085,425.125,177.246,18.974,152.609
C07971=1094.430,239.333,425.099,177.250,18.976,152.609
C07972=1094.435,239.582,425.073,177.253,18.977,152.609
C07973=1094.441,239.831,425.046,177.256,18.979,152.609
C07974=1094.447,240.080,425.020,177.260,18.981,152.608
C07975=1094.452,240.328,424.993,177.262,18.983,152.608
C07976=1094.458,240.576,424.967,177.266,18.985,152.608
C07977=1094.464,240.825,424.941,177.268,18.986,152.608
C07978=1094.469,241.074,424.914,177.272,18.988,152.608
C07979=1094.475,241.323,424.888,177.275,18.990,152.608
C07980=1094.481,241.571,424.862,177.278,18.991,152.607
C07981=1094.486,241.819,424.835,177.281,18.993,152.607
C07982=1094.492,242.068,424.809,177.284,18.995,152.607
C07983=1094.498,242.317,424.782,177.287,18.996,152.607
C07984=1094.503,242.565,424.756,177.291,18.999,152.607
C07985=1094.509,242.813,424.729,177.293,19.000,152.606
C07986=1094.515,243.062,424.703,177.297,19.002,152.606
C07987=1094.520,243.311,424.677,177.300,19.004,152.606
C07988=1094.526,243.559,424.650,177.303,19.005,152.606
C07989=1094.532,243.807,424.623,177.306,19.007,152.606
C07990=1094.537,244.056,424.597,177.309,19.009,152.606
C07991=1094.543,244.305,424.570,177.312,19.010,152.605
C07992=1094.548,244.553,424.543,177.316,19.013,152.605
C07993=1094.554,244.802,424.517,177.318,19.014,152.605
C07994=1094.560,245.050,424.490,177.322,19.016,152.605
C07995=1094.565,245.299,424.464,177.325,19.018,152.605
C07996=1094.570,245.548,424.437,177.328,19.019,152.605
C07997=1094.576,245.796,424.410,177.331,19.021,152.604
C07998=1094.582,246.045,424.384,177.335,19.023,152.604
C07999=1094.588,246.293,424.357,177.337,19.024,152.604
C08000=1094.593,246.541,424.330,177.341,19.027,152.604
C08001=1094.598,246.790,424.303,177.343,19.028,152.604
C08002=1094.604,247.038,424.276,177.347,19.030,152.604
C08003=1094.610,247.287,424.250,177.350,19.032,152.603
C08004=1094.616,247.535,424.223,177.353,19.033,152.603
C08005=1094.621,247.784,424.196,177.356,19.035,152.603
C08006=1094.627,248.033,424.169,177.360,19.037,152.603
C08007=1094.632,248.281,424.142,177.362,19.039,152.603
C08008=1094.638,248.530,424.115,177.365,19.041,152.603
C08009=1094.644,248.778,424.088,177.369,19.043,152.602
C08010=1094.651,249.142,424.049,177.373,19.046,152.602
C08011=1094.659,249.506,424.010,177.378,19.048,152.602
C08012=1094.667,249.870,423.970,177.382,19.051,152.602
C08013=1094.676,250.234,423.931,177.387,19.053,152.602
C08014=1094.681,250.483,423.903,177.390,19.056,152.602
C08015=1094.686,250.731,423.877,177.394,19.057,152.601
C08016=1094.693,250.980,423.850,177.396,19.059,152.601
C08017=1094.698,251.228,423.822,177.399,19.061,152.601
C08018=1094.704,251.476,423.795,177.403,19.063,152.601
C08019=1094.709,251.725,423.768,177.406,19.064,152.601
C08020=1094.715,251.973,423.741,177.409,19.066,152.601
C08021=1094.720,252.222,423.714,177.412,19.068,152.600
C08022=1094.726,252.470,423.687,177.415,19.070,152.600
C08023=1094.731,252.719,423.659,177.418,19.072,152.600
C08024=1094.737,252.968,423.632,177.422,19.074,152.600
C08025=1094.742,253.216,423.605,177.425,19.076,152.600
C08026=1094.748,253.464,423.578,177.428,19.077,152.600
C08027=1094.753,253.713,423.551,177.431,19.080,152.600
C08028=1094.759,253.961,423.524,177.435,19.081,152.599
C08029=1094.765,254.210,423.496,177.437,19.083,152.599
C08030=1094.771,254.458,423.469,177.440,19.085,152.599
C08031=1094.776,254.707,423.442,177.444,19.087,152.599
C08032=1094.782,254.955,423.414,177.446,19.088,152.599
C08033=1094.787,255.203,423.387,177.450,19.091,152.599
C08034=1094.793,255.452,423.360,177.453,19.092,152.598
C08035=1094.799,255.700,423.332,177.457,19.095,152.598
C08036=1094.804,255.949,423.305,177.459,19.096,152.598
C08037=1094.810,256.197,423.278,177.463,19.098,152.598
C08038=1094.815,256.446,423.250,177.466,19.100,152.598
C08039=1094.821,256.695,423.223,177.469,19.101,152.598
C08040=1094.827,256.943,423.195,177.472,19.103,152.598
C08041=1094.833,257.192,423.168,177.475,19.106,152.597
C08042=1094.838,257.440,423.140,177.479,19.107,152.597
C08043=1094.843,257.688,423.113,177.481,19.109,152.597
C08044=1094.849,257.936,423.086,177.485,19.111,152.597
C08045=1094.855,258.185,423.058,177.488,19.113,152.597
C08046=1094.861,258.433,423.031,177.491,19.115,152.597
C08047=1094.866,258.681,423.003,177.494,19.116,152.596
C08048=1094.872,258.931,422.975,177.498,19.119,152.596
C08049=1094.878,259.178,422.948,177.501,19.121,152.596
C08050=1094.883,259.427,422.921,177.504,19.122,152.596
C08051=1094.889,259.676,422.892,177.507,19.124,152.596
C08052=1094.895,259.924,422.865,177.511,19.126,152.596
C08053=1094.900,260.172,422.838,177.514,19.128,152.596
C08054=1094.907,260.421,422.810,177.516,19.130,152.596
C08055=1094.912,260.669,422.782,177.520,19.131,152.595
C08056=1094.918,260.918,422.754,177.523,19.134,152.595
C08057=1094.924,261.166,422.727,177.526,19.135,152.595
C08058=1094.929,261.414,422.699,177.529,19.137,152.595
C08059=1094.935,261.663,422.671,177.533,19.139,152.595
C08060=1094.940,261.911,422.643,177.536,19.141,152.594
C08061=1094.947,262.160,422.616,177.539,19.143,152.594
C08062=1094.955,262.520,422.575,177.544,19.145,152.594
C08063=1094.963,262.881,422.535,177.548,19.148,152.594
C08064=1094.972,263.243,422.494,177.553,19.151,152.594
C08065=1094.980,263.604,422.454,177.557,19.154,152.594
C08066=1094.986,263.852,422.426,177.561,19.155,152.593
C08067=1094.992,264.101,422.399,177.564,19.158,152.593
C08068=1094.997,264.349,422.371,177.567,19.159,152.593
C08069=1095.003,264.598,422.342,177.570,19.161,152.593
C08070=1095.008,264.846,422.314,177.574,19.163,152.593
C08071=1095.014,265.094,422.286,177.577,19.165,152.593
C08072=1095.020,265.343,422.258,177.580,19.168,152.593
C08073=1095.025,265.591,422.230,177.583,19.169,152.593
C08074=1095.031,265.839,422.202,177.586,19.171,152.592
C08075=1095.037,266.087,422.174,177.590,19.173,152.592
C08076=1095.043,266.336,422.146,177.593,19.175,152.592
C08077=1095.048,266.584,422.118,177.595,19.177,152.592
C08078=1095.054,266.832,422.090,177.599,19.179,152.592
C08079=1095.060,267.081,422.062,177.602,19.181,152.592
C08080=1095.065,267.329,422.034,177.606,19.183,152.592
C08081=1095.071,267.577,422.006,177.609,19.185,152.591
C08082=1095.076,267.826,421.978,177.611,19.187,152.591
C08083=1095.082,268.074,421.949,177.615,19.189,152.591
C08084=1095.087,268.322,421.921,177.618,19.191,152.591
C08085=1095.093,268.571,421.893,177.622,19.193,152.591
C08086=1095.099,268.819,421.865,177.625,19.195,152.591
C08087=1095.105,269.068,421.837,177.627,19.197,152.591
C08088=1095.110,269.315,421.808,177.631,19.199,152.591
C08089=1095.116,269.564,421.780,177.634,19.201,152.590
C08090=1095.121,269.812,421.751,177.638,19.203,152.590
C08091=1095.127,270.061,421.723,177.641,19.205,152.590
C08092=1095.132,270.309,421.695,177.643,19.207,152.590
C08093=1095.138,270.557,421.666,177.647,19.209,152.590
C08094=1095.144,270.805,421.638,177.650,19.211,152.590
C08095=1095.150,271.054,421.610,177.653,19.213,152.590
C08096=1095.156,271.303,421.581,177.657,19.216,152.590
C08097=1095.161,271.551,421.553,177.659,19.217,152.590
C08098=1095.166,271.799,421.524,177.663,19.219,152.590
C08099=1095.172,272.047,421.496,177.666,19.221,152.589
C08100=1095.178,272.296,421.467,177.669,19.223,152.589
C08101=1095.183,272.544,421.439,177.673,19.226,152.589
C08102=1095.189,272.792,421.410,177.675,19.227,152.589
C08103=1095.195,273.040,421.382,177.678,19.229,152.589
C08104=1095.200,273.289,421.353,177.682,19.232,152.589
C08105=1095.206,273.538,421.325,177.685,19.234,152.589
C08106=1095.212,273.785,421.296,177.689,19.235,152.589
C08107=1095.218,274.034,421.268,177.692,19.238,152.589
C08108=1095.222,274.282,421.239,177.694,19.239,152.588
C08109=1095.229,274.530,421.210,177.698,19.242,152.588
C08110=1095.235,274.779,421.182,177.701,19.244,152.588
C08111=1095.240,275.026,421.153,177.704,19.246,152.588
C08112=1095.245,275.276,421.124,177.708,19.248,152.588
C08113=1095.251,275.523,421.095,177.711,19.250,152.588
C08114=1095.259,275.888,421.053,177.715,19.253,152.588
C08115=1095.267,276.251,421.011,177.720,19.256,152.588
C08116=1095.276,276.615,420.968,177.725,19.260,152.588
C08117=1095.284,276.979,420.927,177.729,19.262,152.588
C08118=1095.290,277.227,420.898,177.732,19.265,152.587
C08119=1095.296,277.475,420.869,177.736,19.267,152.587
C08120=1095.301,277.724,420.840,177.739,19.269,152.587
C08121=1095.307,277.972,420.811,177.742,19.271,152.587
C08122=1095.312,278.220,420.783,177.745,19.273,152.587
C08123=1095.318,278.469,420.753,177.748,19.275,152.587
C08124=1095.324,278.717,420.724,177.752,19.277,152.587
C08125=1095.329,278.965,420.696,177.755,19.279,152.587
C08126=1095.335,279.213,420.667,177.758,19.282,152.587
C08127=1095.341,279.461,420.638,177.761,19.284,152.587
C08128=1095.346,279.709,420.608,177.765,19.286,152.587
C08129=1095.352,279.958,420.580,177.767,19.288,152.586
C08130=1095.358,280.206,420.550,177.770,19.290,152.587
C08131=1095.364,280.454,420.521,177.774,19.292,152.586
C08132=1095.369,280.702,420.492,177.777,19.295,152.586
C08133=1095.375,280.951,420.464,177.780,19.297,152.586
C08134=1095.380,281.199,420.434,177.784,19.299,152.586
C08135=1095.387,281.447,420.405,177.787,19.301,152.586
C08136=1095.391,281.695,420.376,177.790,19.303,152.586
C08137=1095.398,281.943,420.347,177.794,19.306,152.586
C08138=1095.403,282.192,420.317,177.796,19.307,152.586
C08139=1095.408,282.440,420.289,177.799,19.309,152.586
C08140=1095.414,282.688,420.260,177.802,19.312,152.586
C08141=1095.420,282.937,420.230,177.806,19.314,152.586
C08142=1095.426,283.185,420.201,177.809,19.316,152.586
C08143=1095.431,283.433,420.172,177.812,19.319,152.586
C08144=1095.436,283.681,420.142,177.816,19.321,152.585
C08145=1095.442,283.929,420.113,177.819,19.323,152.585
C08146=1095.448,284.178,420.083,177.822,19.326,152.585
C08147=1095.453,284.425,420.054,177.825,19.327,152.585
C08148=1095.459,284.673,420.025,177.828,19.329,152.585
C08149=1095.465,284.922,419.995,177.831,19.332,152.585
C08150=1095.470,285.170,419.966,177.835,19.334,152.585
C08151=1095.476,285.418,419.937,177.838,19.336,152.585
C08152=1095.481,285.666,419.907,177.841,19.339,152.585
C08153=1095.487,285.915,419.878,177.844,19.341,152.585
C08154=1095.493,286.163,419.849,177.848,19.343,152.585
C08155=1095.499,286.411,419.819,177.851,19.346,152.585
C08156=1095.504,286.659,419.789,177.854,19.348,152.585
C08157=1095.510,286.907,419.759,177.857,19.350,152.585
C08158=1095.516,287.156,419.730,177.861,19.352,152.585
C08159=1095.521,287.403,419.701,177.863,19.354,152.585
C08160=1095.527,287.652,419.671,177.866,19.357,152.585
C08161=1095.533,287.900,419.642,177.869,19.359,152.585
C08162=1095.539,288.148,419.612,177.873,19.361,152.584
C08163=1095.544,288.396,419.582,177.876,19.363,152.584
C08164=1095.550,288.645,419.553,177.879,19.365,152.584
C08165=1095.556,288.893,419.523,177.882,19.368,152.584
C08166=1095.565,289.265,419.478,177.887,19.371,152.584
C08167=1095.573,289.639,419.434,177.892,19.375,152.584
C08168=1095.581,290.012,419.389,177.897,19.378,152.584
C08169=1095.589,290.385,419.344,177.902,19.382,152.584
C08170=1095.595,290.634,419.315,177.905,19.384,152.584
C08171=1095.601,290.881,419.284,177.909,19.386,152.584
C08172=1095.606,291.130,419.255,177.912,19.389,152.584
C08173=1095.613,291.378,419.226,177.915,19.391,152.584
C08174=1095.618,291.626,419.195,177.918,19.393,152.584
C08175=1095.624,291.874,419.166,177.921,19.396,152.584
C08176=1095.630,292.122,419.135,177.924,19.398,152.584
C08177=1095.635,292.371,419.106,177.927,19.400,152.584
C08178=1095.641,292.618,419.075,177.930,19.403,152.584
C08179=1095.647,292.867,419.046,177.933,19.405,152.584
C08180=1095.652,293.115,419.015,177.937,19.407,152.584
C08181=1095.658,293.363,418.986,177.940,19.410,152.584
C08182=1095.664,293.611,418.955,177.943,19.412,152.584
C08183=1095.669,293.859,418.926,177.946,19.414,152.584
C08184=1095.674,294.106,418.896,177.950,19.417,152.584
C08185=1095.680,294.355,418.866,177.953,19.419,152.584
C08186=1095.686,294.603,418.836,177.956,19.421,152.584
C08187=1095.691,294.851,418.806,177.959,19.424,152.584
C08188=1095.697,295.099,418.776,177.962,19.426,152.584
C08189=1095.704,295.347,418.745,177.965,19.429,152.584
C08190=1095.709,295.596,418.715,177.969,19.431,152.584
C08191=1095.715,295.844,418.685,177.972,19.433,152.583
C08192=1095.721,296.092,418.655,177.975,19.436,152.584
C08193=1095.726,296.340,418.625,177.978,19.438,152.583
C08194=1095.732,296.588,418.595,177.982,19.441,152.584
C08195=1095.737,296.836,418.564,177.985,19.443,152.583
C08196=1095.743,297.084,418.534,177.988,19.446,152.584
C08197=1095.748,297.332,418.504,177.991,19.448,152.583
C08198=1095.754,297.580,418.473,177.994,19.450,152.584
C08199=1095.760,297.828,418.443,177.997,19.453,152.584
C08200=1095.766,298.076,418.413,178.001,19.455,152.583
C08201=1095.771,298.324,418.383,178.004,19.458,152.584
C08202=1095.776,298.572,418.352,178.007,19.460,152.583
C08203=1095.782,298.820,418.322,178.010,19.463,152.584
C08204=1095.788,299.068,418.291,178.013,19.465,152.584
C08205=1095.793,299.316,418.261,178.016,19.468,152.584
C08206=1095.799,299.564,418.231,178.020,19.470,152.584
C08207=1095.804,299.812,418.201,178.023,19.473,152.584
C08208=1095.810,300.060,418.170,178.026,19.475,152.584
C08209=1095.815,300.308,418.139,178.030,19.478,152.584
C08210=1095.821,300.556,418.109,178.033,19.481,152.584
C08211=1095.826,300.804,418.078,178.036,19.484,152.584
C08212=1095.832,301.052,418.048,178.039,19.486,152.584
C08213=1095.838,301.301,418.016,178.043,19.488,152.584
C08214=1095.844,301.549,417.986,178.046,19.491,152.584
C08215=1095.849,301.796,417.956,178.049,19.494,152.584
C08216=1095.854,302.045,417.925,178.052,19.496,152.584
C08217=1095.860,302.292,417.894,178.055,19.499,152.584
C08218=1095.869,302.679,417.847,178.060,19.503,152.584
C08219=1095.878,303.067,417.798,178.065,19.507,152.584
C08220=1095.886,303.454,417.751,178.070,19.511,152.584
C08221=1095.895,303.841,417.703,178.075,19.514,152.584
C08222=1095.901,304.090,417.672,178.078,19.517,152.584
C08223=1095.907,304.337,417.641,178.082,19.520,152.584
C08224=1095.912,304.585,417.610,178.085,19.523,152.584
C08225=1095.918,304.833,417.579,178.088,19.525,152.584
C08226=1095.924,305.081,417.549,178.091,19.528,152.584
C08227=1095.929,305.329,417.518,178.094,19.530,152.584
C08228=1095.935,305.577,417.487,178.097,19.533,152.584
C08229=1095.940,305.825,417.456,178.100,19.536,152.584
C08230=1095.946,306.073,417.425,178.103,19.538,152.585
C08231=1095.951,306.321,417.394,178.106,19.541,152.585
C08232=1095.957,306.569,417.364,178.110,19.544,152.585
C08233=1095.963,306.817,417.332,178.113,19.546,152.585
C08234=1095.969,307.065,417.302,178.116,19.548,152.585
C08235=1095.974,307.313,417.271,178.120,19.552,152.585
C08236=1095.981,307.561,417.239,178.123,19.554,152.585
C08237=1095.986,307.809,417.208,178.126,19.557,152.585
C08238=1095.991,308.057,417.177,178.129,19.559,152.585
C08239=1095.997,308.304,417.146,178.132,19.562,152.585
C08240=1096.003,308.553,417.115,178.135,19.565,152.585
C08241=1096.009,308.801,417.085,178.138,19.567,152.585
C08242=1096.014,309.048,417.053,178.142,19.570,152.585
C08243=1096.020,309.297,417.022,178.145,19.572,152.585
C08244=1096.026,309.544,416.991,178.149,19.575,152.585
C08245=1096.031,309.792,416.960,178.152,19.578,152.585
C08246=1096.038,310.040,416.928,178.155,19.581,152.585
C08247=1096.043,310.288,416.897,178.158,19.583,152.585
C08248=1096.049,310.536,416.866,178.161,19.586,152.585
C08249=1096.054,310.784,416.835,178.164,19.589,152.586
C08250=1096.060,311.032,416.803,178.167,19.591,152.586
C08251=1096.066,311.280,416.773,178.170,19.594,152.586
C08252=1096.072,311.528,416.741,178.173,19.596,152.586
C08253=1096.077,311.776,416.710,178.177,19.600,152.586
C08254=1096.083,312.024,416.678,178.180,19.602,152.586
C08255=1096.089,312.272,416.647,178.183,19.605,152.586
C08256=1096.095,312.520,416.616,178.186,19.608,152.586
C08257=1096.101,312.768,416.584,178.190,19.610,152.586
C08258=1096.106,313.015,416.553,178.193,19.613,152.586
C08259=1096.112,313.264,416.522,178.196,19.615,152.586
C08260=1096.118,313.511,416.490,178.199,19.618,152.586
C08261=1096.124,313.759,416.458,178.203,19.621,152.586
C08262=1096.130,314.007,416.428,178.206,19.624,152.586
C08263=1096.136,314.255,416.396,178.209,19.627,152.587
C08264=1096.141,314.503,416.364,178.212,19.629,152.587
C08265=1096.147,314.752,416.333,178.215,19.632,152.587
C08266=1096.153,314.999,416.302,178.218,19.634,152.587
C08267=1096.159,315.247,416.270,178.221,19.637,152.587
C08268=1096.164,315.495,416.238,178.225,19.641,152.587
C08269=1096.170,315.743,416.206,178.228,19.643,152.587
C08270=1096.179,316.133,416.157,178.232,19.647,152.587
C08271=1096.187,316.522,416.107,178.238,19.652,152.587
C08272=1096.196,316.912,416.057,178.242,19.657,152.588
C08273=1096.205,317.301,416.007,178.247,19.662,152.588
C08274=1096.211,317.550,415.975,178.251,19.664,152.588
C08275=1096.216,317.797,415.944,178.253,19.667,152.588
C08276=1096.222,318.045,415.911,178.257,19.670,152.588
C08277=1096.227,318.293,415.880,178.260,19.673,152.588
C08278=1096.233,318.542,415.849,178.263,19.676,152.589
C08279=1096.238,318.789,415.817,178.266,19.679,152.589
C08280=1096.244,319.038,415.784,178.269,19.682,152.589
C08281=1096.249,319.285,415.753,178.273,19.685,152.589
C08282=1096.255,319.534,415.721,178.276,19.688,152.589
C08283=1096.260,319.781,415.689,178.279,19.691,152.589
C08284=1096.267,320.029,415.656,178.282,19.694,152.589
C08285=1096.272,320.276,415.624,178.285,19.696,152.590
C08286=1096.278,320.524,415.592,178.289,19.700,152.590
C08287=1096.284,320.772,415.561,178.292,19.703,152.590
C08288=1096.289,321.020,415.528,178.295,19.706,152.590
C08289=1096.294,321.268,415.496,178.298,19.708,152.590
C08290=1096.300,321.516,415.464,178.300,19.711,152.590
C08291=1096.306,321.764,415.432,178.304,19.715,152.590
C08292=1096.312,322.012,415.401,178.307,19.718,152.591
C08293=1096.318,322.259,415.368,178.310,19.721,152.591
C08294=1096.322,322.507,415.336,178.313,19.723,152.591
C08295=1096.328,322.756,415.304,178.316,19.727,152.591
C08296=1096.334,323.004,415.272,178.320,19.730,152.591
C08297=1096.340,323.251,415.240,178.323,19.733,152.591
C08298=1096.346,323.499,415.207,178.326,19.735,152.591
C08299=1096.351,323.747,415.175,178.329,19.738,152.592
C08300=1096.357,323.995,415.143,178.332,19.742,152.592
C08301=1096.363,324.242,415.110,178.336,19.745,152.592
C08302=1096.368,324.490,415.079,178.338,19.748,152.592
C08303=1096.374,324.738,415.047,178.341,19.751,152.592
C08304=1096.380,324.986,415.013,178.345,19.754,152.592
C08305=1096.386,325.234,414.981,178.348,19.757,152.593
C08306=1096.391,325.482,414.950,178.351,19.760,152.593
C08307=1096.397,325.730,414.916,178.354,19.763,152.593
C08308=1096.403,325.978,414.884,178.358,19.766,152.593
C08309=1096.408,326.225,414.853,178.360,19.770,152.593
C08310=1096.415,326.473,414.820,178.364,19.772,152.594
C08311=1096.420,326.722,414.787,178.366,19.775,152.594
C08312=1096.426,326.969,414.754,178.370,19.779,152.594
C08313=1096.431,327.217,414.723,178.373,19.782,152.594
C08314=1096.437,327.465,414.689,178.376,19.785,152.594
C08315=1096.443,327.713,414.657,178.380,19.788,152.594
C08316=1096.449,327.960,414.625,178.383,19.791,152.595
C08317=1096.455,328.208,414.593,178.385,19.794,152.595
C08318=1096.460,328.456,414.560,178.389,19.797,152.595
C08319=1096.466,328.704,414.528,178.392,19.801,152.595
C08320=1096.473,328.952,414.495,178.395,19.804,152.595
C08321=1096.478,329.200,414.462,178.398,19.807,152.596
C08322=1096.487,329.582,414.412,178.403,19.811,152.596
C08323=1096.496,329.965,414.361,178.408,19.817,152.596
C08324=1096.505,330.347,414.311,178.413,19.821,152.596
C08325=1096.514,330.731,414.260,178.418,19.826,152.597
C08326=1096.520,330.978,414.228,178.421,19.829,152.597
C08327=1096.526,331.225,414.195,178.423,19.832,152.597
C08328=1096.531,331.473,414.162,178.427,19.836,152.597
C08329=1096.537,331.721,414.130,178.430,19.839,152.598
C08330=1096.543,331.969,414.096,178.433,19.842,152.598
C08331=1096.549,332.217,414.064,178.437,19.845,152.598
C08332=1096.554,332.465,414.030,178.439,19.849,152.598
C08333=1096.561,332.712,413.998,178.442,19.852,152.599
C08334=1096.566,332.961,413.965,178.446,19.856,152.599
C08335=1096.571,333.208,413.932,178.449,19.859,152.599
C08336=1096.577,333.456,413.899,178.452,19.862,152.599
C08337=1096.583,333.704,413.866,178.455,19.865,152.599
C08338=1096.588,333.952,413.833,178.458,19.869,152.600
C08339=1096.595,334.199,413.800,178.462,19.872,152.600
C08340=1096.600,334.447,413.767,178.465,19.875,152.600
C08341=1096.606,334.695,413.733,178.467,19.879,152.600
C08342=1096.611,334.942,413.701,178.471,19.882,152.601
C08343=1096.617,335.190,413.668,178.474,19.886,152.601
C08344=1096.622,335.438,413.635,178.477,19.889,152.601
C08345=1096.629,335.686,413.602,178.480,19.892,152.602
C08346=1096.634,335.934,413.569,178.483,19.895,152.602
C08347=1096.640,336.181,413.535,178.487,19.899,152.602
C08348=1096.646,336.429,413.501,178.489,19.902,152.602
C08349=1096.652,336.677,413.469,178.492,19.906,152.603
C08350=1096.657,336.924,413.435,178.496,19.910,152.603
C08351=1096.663,337.172,413.402,178.499,19.913,152.603
C08352=1096.668,337.420,413.369,178.502,19.916,152.603
C08353=1096.675,337.668,413.336,178.505,19.920,152.604
C08354=1096.680,337.916,413.303,178.508,19.923,152.604
C08355=1096.686,338.164,413.269,178.512,19.926,152.604
C08356=1096.691,338.412,413.236,178.514,19.930,152.605
C08357=1096.698,338.659,413.202,178.518,19.934,152.605
C08358=1096.704,338.906,413.169,178.521,19.937,152.605
C08359=1096.709,339.154,413.136,178.523,19.940,152.605
C08360=1096.715,339.402,413.102,178.527,19.944,152.606
C08361=1096.721,339.650,413.068,178.530,19.947,152.606
C08362=1096.726,339.897,413.035,178.533,19.951,152.606
C08363=1096.732,340.145,413.002,178.536,19.955,152.607
C08364=1096.737,340.393,412.969,178.539,19.958,152.607
C08365=1096.743,340.640,412.935,178.542,19.962,152.607
C08366=1096.749,340.888,412.901,178.545,19.965,152.607
C08367=1096.754,341.136,412.868,178.548,19.969,152.608
C08368=1096.760,341.384,412.834,178.551,19.972,152.608
C08369=1096.766,341.631,412.801,178.555,19.976,152.608
C08370=1096.772,341.879,412.768,178.557,19.980,152.609
C08371=1096.778,342.126,412.733,178.561,19.984,152.609
C08372=1096.783,342.374,412.700,178.564,19.987,152.609
C08373=1096.789,342.622,412.666,178.567,19.991,152.610
C08374=1096.798,342.998,412.615,178.571,19.996,152.610
C08375=1096.806,343.375,412.564,178.576,20.001,152.611
C08376=1096.815,343.751,412.512,178.581,20.007,152.611
C08377=1096.824,344.129,412.461,178.586,20.013,152.612
C08378=1096.830,344.377,412.427,178.588,20.016,152.612
C08379=1096.836,344.624,412.393,178.592,20.020,152.612
C08380=1096.841,344.872,412.360,178.595,20.023,152.613
C08381=1096.847,345.119,412.326,178.598,20.027,152.613
C08382=1096.852,345.367,412.291,178.601,20.031,152.614
C08383=1096.858,345.615,412.258,178.604,20.035,152.614
C08384=1096.864,345.862,412.224,178.607,20.039,152.614
C08385=1096.870,346.109,412.190,178.610,20.043,152.615
C08386=1096.876,346.358,412.156,178.613,20.046,152.615
C08387=1096.882,346.605,412.122,178.617,20.050,152.615
C08388=1096.887,346.853,412.088,178.619,20.054,152.616
C08389=1096.892,347.101,412.054,178.623,20.058,152.616
C08390=1096.898,347.348,412.020,178.625,20.061,152.616
C08391=1096.904,347.595,411.986,178.629,20.065,152.617
C08392=1096.910,347.842,411.952,178.631,20.069,152.617
C08393=1096.915,348.091,411.918,178.635,20.073,152.618
C08394=1096.921,348.339,411.884,178.637,20.077,152.618
C08395=1096.927,348.586,411.850,178.641,20.081,152.618
C08396=1096.933,348.833,411.816,178.644,20.085,152.619
C08397=1096.938,349.081,411.781,178.647,20.088,152.619
C08398=1096.944,349.329,411.746,178.650,20.092,152.620
C08399=1096.950,349.577,411.713,178.653,20.096,152.620
C08400=1096.955,349.824,411.679,178.656,20.100,152.620
C08401=1096.961,350.072,411.644,178.659,20.104,152.621
C08402=1096.967,350.319,411.610,178.662,20.108,152.621
C08403=1096.973,350.567,411.575,178.665,20.112,152.622
C08404=1096.978,350.814,411.541,178.668,20.116,152.622
C08405=1096.984,351.062,411.507,178.672,20.120,152.622
C08406=1096.989,351.309,411.473,178.674,20.124,152.623
C08407=1096.996,351.557,411.438,178.678,20.128,152.623
C08408=1097.002,351.805,411.404,178.680,20.131,152.624
C08409=1097.007,352.052,411.370,178.684,20.136,152.624
C08410=1097.013,352.299,411.335,178.687,20.140,152.625
C08411=1097.019,352.547,411.301,178.690,20.143,152.625
C08412=1097.024,352.795,411.266,178.693,20.148,152.625
C08413=1097.030,353.042,411.232,178.696,20.151,152.626
C08414=1097.036,353.290,411.197,178.699,20.155,152.626
C08415=1097.042,353.537,411.163,178.702,20.159,152.627
C08416=1097.047,353.785,411.128,178.705,20.163,152.627
C08417=1097.053,354.032,411.094,178.708,20.168,152.628
C08418=1097.059,354.280,411.059,178.711,20.171,152.628
C08419=1097.065,354.528,411.025,178.714,20.176,152.629
C08420=1097.070,354.775,410.989,178.717,20.180,152.629
C08421=1097.076,355.023,410.955,178.720,20.184,152.630
C08422=1097.082,355.270,410.920,178.723,20.188,152.630
C08423=1097.087,355.518,410.886,178.725,20.192,152.631
C08424=1097.094,355.765,410.851,178.729,20.196,152.631
C08425=1097.099,356.012,410.817,178.732,20.201,152.631
C08426=1097.108,356.392,410.763,178.737,20.207,152.632
C08427=1097.117,356.770,410.710,178.741,20.213,152.633
C08428=1097.126,357.150,410.656,178.746,20.220,152.634
C08429=1097.135,357.529,410.603,178.750,20.226,152.635
C08430=1097.140,357.777,410.568,178.754,20.230,152.635
C08431=1097.146,358.023,410.533,178.757,20.235,152.635
C08432=1097.152,358.272,410.498,178.759,20.239,152.636
C08433=1097.158,358.518,410.464,178.763,20.243,152.636
C08434=1097.163,358.767,410.429,178.766,20.248,152.637
C08435=1097.169,359.014,410.393,178.768,20.251,152.637
C08436=1097.175,359.261,410.359,178.772,20.256,152.638
C08437=1097.181,359.509,410.323,178.775,20.260,152.638
C08438=1097.186,359.756,410.289,178.777,20.264,152.639
C08439=1097.193,360.004,410.254,178.780,20.269,152.640
C08440=1097.198,360.251,410.218,178.784,20.273,152.640
C08441=1097.204,360.499,410.183,178.786,20.277,152.641
C08442=1097.209,360.746,410.148,178.789,20.282,152.641
C08443=1097.215,360.993,410.114,178.793,20.286,152.642
C08444=1097.221,361.241,410.078,178.795,20.290,152.642
C08445=1097.227,361.488,410.043,178.798,20.295,152.643
C08446=1097.232,361.736,410.008,178.801,20.299,152.643
C08447=1097.238,361.983,409.972,178.805,20.304,152.644
C08448=1097.244,362.231,409.937,178.807,20.308,152.644
C08449=1097.250,362.477,409.902,178.810,20.313,152.645
C08450=1097.256,362.726,409.867,178.813,20.317,152.646
C08451=1097.261,362.973,409.832,178.817,20.322,152.646
C08452=1097.267,363.220,409.796,178.819,20.326,152.647
C08453=1097.273,363.467,409.760,178.822,20.331,152.647
C08454=1097.279,363.715,409.725,178.825,20.335,152.648
C08455=1097.284,363.962,409.691,178.828,20.340,152.648
C08456=1097.290,364.210,409.655,178.831,20.344,152.649
C08457=1097.296,364.457,409.620,178.834,20.349,152.650
C08458=1097.302,364.705,409.584,178.837,20.353,152.650
C08459=1097.307,364.952,409.548,178.840,20.358,152.651
C08460=1097.313,365.199,409.513,178.843,20.362,152.651
C08461=1097.319,365.446,409.477,178.846,20.367,152.652
C08462=1097.325,365.694,409.442,178.849,20.371,152.653
C08463=1097.331,365.942,409.406,178.852,20.376,152.653
C08464=1097.336,366.189,409.371,178.854,20.380,152.654
C08465=1097.342,366.436,409.335,178.857,20.385,152.654
C08466=1097.348,366.683,409.299,178.861,20.390,152.655
C08467=1097.354,366.931,409.264,178.864,20.395,152.656
C08468=1097.359,367.178,409.228,178.867,20.400,152.656
C08469=1097.365,367.426,409.193,178.869,20.404,152.657
C08470=1097.371,367.672,409.157,178.872,20.409,152.658
C08471=1097.377,367.920,409.122,178.875,20.414,152.658
C08472=1097.382,368.167,409.086,178.878,20.418,152.659
C08473=1097.388,368.414,409.049,178.881,20.423,152.659
C08474=1097.394,368.662,409.013,178.884,20.427,152.660
C08475=1097.399,368.909,408.978,178.887,20.432,152.661
C08476=1097.405,369.157,408.942,178.890,20.437,152.661
C08477=1097.411,369.404,408.907,178.893,20.442,152.662
C08478=1097.420,369.798,408.849,178.897,20.450,152.663
C08479=1097.430,370.193,408.792,178.901,20.457,152.664
C08480=1097.439,370.586,408.735,178.906,20.465,152.665
C08481=1097.448,370.981,408.677,178.911,20.473,152.666
C08482=1097.453,371.228,408.642,178.914,20.478,152.667
C08483=1097.460,371.475,408.606,178.916,20.483,152.668
C08484=1097.466,371.723,408.570,178.919,20.487,152.669
C08485=1097.471,371.969,408.533,178.922,20.492,152.669
C08486=1097.477,372.217,408.497,178.926,20.497,152.670
C08487=1097.483,372.465,408.462,178.928,20.502,152.671
C08488=1097.489,372.712,408.425,178.931,20.507,152.671
C08489=1097.495,372.959,408.390,178.935,20.512,152.672
C08490=1097.500,373.206,408.353,178.937,20.517,152.673
C08491=1097.506,373.454,408.317,178.940,20.522,152.673
C08492=1097.512,373.701,408.281,178.943,20.527,152.674
C08493=1097.518,373.948,408.245,178.946,20.532,152.675
C08494=1097.523,374.195,408.208,178.949,20.537,152.676
C08495=1097.530,374.443,408.173,178.951,20.542,152.676
C08496=1097.535,374.689,408.137,178.954,20.547,152.677
C08497=1097.541,374.936,408.099,178.957,20.552,152.678
C08498=1097.547,375.184,408.064,178.960,20.557,152.679
C08499=1097.552,375.432,408.027,178.963,20.563,152.679
C08500=1097.558,375.678,407.991,178.966,20.568,152.680
C08501=1097.564,375.926,407.954,178.969,20.573,152.681
C08502=1097.570,376.173,407.918,178.971,20.578,152.682
C08503=1097.575,376.420,407.881,178.974,20.583,152.683
C08504=1097.581,376.667,407.845,178.977,20.588,152.683
C08505=1097.586,376.915,407.808,178.980,20.593,152.684
C08506=1097.593,377.162,407.772,178.983,20.599,152.685
C08507=1097.598,377.409,407.735,178.985,20.604,152.686
C08508=1097.604,377.656,407.700,178.988,20.609,152.687
C08509=1097.609,377.903,407.663,178.991,20.615,152.687
C08510=1097.616,378.150,407.626,178.994,20.620,152.688
C08511=1097.621,378.398,407.589,178.997,20.625,152.689
C08512=1097.628,378.645,407.553,179.000,20.630,152.690
C08513=1097.633,378.892,407.516,179.003,20.636,152.691
C08514=1097.639,379.139,407.479,179.005,20.641,152.691
C08515=1097.645,379.386,407.442,179.008,20.646,152.692
C08516=1097.651,379.634,407.407,179.011,20.652,152.693
C08517=1097.656,379.881,407.370,179.014,20.657,152.694
C08518=1097.663,380.128,407.333,179.017,20.663,152.695
C08519=1097.668,380.375,407.296,179.020,20.668,152.695
C08520=1097.673,380.622,407.260,179.022,20.673,152.696
C08521=1097.680,380.869,407.223,179.025,20.679,152.697
C08522=1097.685,381.116,407.185,179.028,20.684,152.698
C08523=1097.692,381.363,407.149,179.031,20.689,152.699
C08524=1097.697,381.610,407.112,179.034,20.695,152.700
C08525=1097.703,381.858,407.075,179.036,20.700,152.701
C08526=1097.709,382.105,407.038,179.039,20.706,152.702
C08527=1097.715,382.352,407.001,179.042,20.711,152.702
C08528=1097.721,382.599,406.965,179.045,20.717,152.703
C08529=1097.727,382.846,406.928,179.047,20.722,152.704
C08530=1097.731,383.057,406.896,179.050,20.727,152.705
C08531=1097.737,383.268,406.865,179.052,20.732,152.706
C08532=1097.741,383.478,406.833,179.054,20.737,152.706
C08533=1097.746,383.688,406.801,179.058,20.742,152.707
C08534=1097.752,383.899,406.770,179.060,20.746,152.708
C08535=1097.757,384.110,406.738,179.062,20.751,152.709
C08536=1097.761,384.321,406.706,179.065,20.756,152.710
C08537=1097.766,384.532,406.674,179.067,20.761,152.710
C08538=1097.772,384.779,406.638,179.069,20.767,152.711
C08539=1097.777,385.025,406.601,179.072,20.773,152.712
C08540=1097.783,385.272,406.563,179.075,20.778,152.713
C08541=1097.789,385.520,406.526,179.077,20.784,152.714
C08542=1097.794,385.767,406.489,179.080,20.790,152.715
C08543=1097.800,386.014,406.451,179.083,20.796,152.716
C08544=1097.806,386.261,406.414,179.086,20.802,152.717
C08545=1097.812,386.508,406.377,179.089,20.807,152.718
C08546=1097.818,386.755,406.340,179.091,20.813,152.719
C08547=1097.824,387.002,406.302,179.094,20.819,152.720
C08548=1097.830,387.249,406.265,179.097,20.825,152.721
C08549=1097.835,387.496,406.228,179.099,20.830,152.722
C08550=1097.841,387.743,406.191,179.102,20.836,152.723
C08551=1097.847,387.990,406.153,179.105,20.843,152.724
C08552=1097.853,388.237,406.116,179.108,20.848,152.725
C08553=1097.859,388.484,406.078,179.111,20.854,152.726
C08554=1097.864,388.731,406.041,179.113,20.860,152.727
C08555=1097.870,388.978,406.003,179.116,20.866,152.728
C08556=1097.877,389.225,405.965,179.118,20.872,152.729
C08557=1097.882,389.473,405.928,179.122,20.878,152.730
C08558=1097.888,389.720,405.890,179.124,20.884,152.731
C08559=1097.894,389.966,405.853,179.127,20.890,152.732
C08560=1097.900,390.214,405.816,179.129,20.896,152.733
C08561=1097.906,390.460,405.778,179.132,20.902,152.734
C08562=1097.911,390.707,405.740,179.135,20.908,152.735
C08563=1097.917,390.954,405.702,179.138,20.915,152.736
C08564=1097.924,391.202,405.665,179.140,20.921,152.737
C08565=1097.929,391.449,405.627,179.143,20.926,152.738
C08566=1097.935,391.695,405.589,179.146,20.932,152.739
C08567=1097.941,391.942,405.552,179.149,20.939,152.740
C08568=1097.947,392.189,405.514,179.151,20.945,152.741
C08569=1097.953,392.437,405.477,179.154,20.951,152.742
C08570=1097.959,392.684,405.439,179.156,20.957,152.743
C08571=1097.965,392.931,405.401,179.160,20.964,152.744
C08572=1097.970,393.178,405.363,179.162,20.970,152.746
C08573=1097.976,393.424,405.325,179.165,20.976,152.747
C08574=1097.982,393.671,405.287,179.167,20.983,152.748
C08575=1097.989,393.918,405.249,179.170,20.989,152.749
C08576=1097.994,394.166,405.211,179.173,20.995,152.750
C08577=1098.000,394.412,405.173,179.175,21.002,152.751
C08578=1098.006,394.659,405.135,179.178,21.008,152.752
C08579=1098.012,394.906,405.097,179.181,21.015,152.753
C08580=1098.017,395.154,405.059,179.183,21.021,152.755
C08581=1098.023,395.400,405.021,179.186,21.027,152.756
C08582=1098.029,395.647,404.983,179.189,21.034,152.757
C08583=1098.035,395.895,404.944,179.191,21.040,152.758
C08584=1098.041,396.142,404.907,179.194,21.047,152.759
C08585=1098.047,396.388,404.869,179.196,21.053,152.760
C08586=1098.052,396.605,404.835,179.199,21.059,152.761
C08587=1098.057,396.823,404.801,179.201,21.065,152.762
C08588=1098.063,397.039,404.768,179.203,21.071,152.764
C08589=1098.067,397.256,404.734,179.206,21.076,152.765
C08590=1098.072,397.473,404.700,179.208,21.082,152.766
C08591=1098.078,397.690,404.667,179.211,21.089,152.767
C08592=1098.083,397.907,404.634,179.212,21.094,152.768
C08593=1098.088,398.124,404.600,179.215,21.100,152.769
C08594=1098.094,398.371,404.562,179.217,21.107,152.770
C08595=1098.100,398.618,404.522,179.220,21.114,152.771
C08596=1098.106,398.865,404.485,179.222,21.120,152.773
C08597=1098.111,399.112,404.446,179.225,21.127,152.774
C08598=1098.117,399.359,404.408,179.228,21.134,152.775
C08599=1098.123,399.606,404.369,179.230,21.140,152.776
C08600=1098.129,399.853,404.331,179.233,21.147,152.777
C08601=1098.135,400.100,404.292,179.236,21.154,152.779
C08602=1098.141,400.346,404.254,179.238,21.161,152.780
C08603=1098.146,400.594,404.215,179.241,21.168,152.781
C08604=1098.152,400.841,404.176,179.243,21.175,152.783
C08605=1098.158,401.088,404.138,179.246,21.182,152.784
C08606=1098.164,401.335,404.099,179.248,21.189,152.785
C08607=1098.170,401.581,404.061,179.251,21.196,152.786
C08608=1098.176,401.828,404.022,179.254,21.203,152.788
C08609=1098.181,402.075,403.984,179.256,21.209,152.789
C08610=1098.188,402.322,403.945,179.259,21.217,152.790
C08611=1098.193,402.569,403.906,179.261,21.223,152.792
C08612=1098.199,402.816,403.867,179.264,21.231,152.793
C08613=1098.205,403.063,403.829,179.266,21.238,152.794
C08614=1098.211,403.310,403.790,179.269,21.245,152.796
C08615=1098.217,403.557,403.751,179.271,21.252,152.797
C08616=1098.223,403.804,403.712,179.274,21.260,152.798
C08617=1098.229,404.051,403.674,179.276,21.267,152.800
C08618=1098.235,404.298,403.634,179.279,21.274,152.801
C08619=1098.241,404.544,403.596,179.281,21.281,152.802
C08620=1098.247,404.791,403.556,179.284,21.288,152.804
C08621=1098.252,405.038,403.518,179.287,21.295,152.805
C08622=1098.258,405.285,403.478,179.289,21.303,152.807
C08623=1098.264,405.532,403.439,179.292,21.311,152.808
C08624=1098.270,405.779,403.401,179.294,21.317,152.809
C08625=1098.276,406.025,403.362,179.297,21.325,152.811
C08626=1098.282,406.273,403.323,179.299,21.332,152.812
C08627=1098.288,406.520,403.283,179.302,21.340,152.814
C08628=1098.293,406.766,403.244,179.304,21.347,152.815
C08629=1098.299,407.013,403.205,179.307,21.355,152.817
C08630=1098.305,407.260,403.166,179.310,21.363,152.818
C08631=1098.311,407.507,403.126,179.312,21.370,152.820
C08632=1098.317,407.753,403.088,179.315,21.377,152.821
C08633=1098.323,408.000,403.048,179.318,21.385,152.822
C08634=1098.329,408.247,403.009,179.320,21.393,152.824
C08635=1098.335,408.494,402.970,179.322,21.400,152.825
C08636=1098.341,408.741,402.931,179.325,21.408,152.827
C08637=1098.346,408.987,402.891,179.327,21.416,152.828
C08638=1098.352,409.235,402.851,179.330,21.423,152.830
C08639=1098.358,409.482,402.812,179.333,21.432,152.832
C08640=1098.363,409.728,402.772,179.335,21.439,152.833
C08641=1098.369,409.975,402.733,179.337,21.447,152.835
C08642=1098.375,410.192,402.699,179.339,21.454,152.836
C08643=1098.380,410.410,402.663,179.342,21.461,152.837
C08644=1098.385,410.627,402.629,179.344,21.468,152.839
C08645=1098.391,410.844,402.595,179.346,21.474,152.840
C08646=1098.395,411.061,402.559,179.348,21.481,152.841
C08647=1098.401,411.277,402.525,179.350,21.489,152.843
C08648=1098.406,411.495,402.490,179.352,21.495,152.844
C08649=1098.411,411.712,402.455,179.355,21.502,152.846
C08650=1098.417,411.959,402.415,179.357,21.511,152.847
C08651=1098.423,412.206,402.376,179.360,21.518,152.849
C08652=1098.429,412.452,402.337,179.363,21.527,152.850
C08653=1098.434,412.699,402.296,179.365,21.535,152.852
C08654=1098.440,412.946,402.257,179.367,21.543,152.854
C08655=1098.447,413.193,402.216,179.370,21.551,152.855
C08656=1098.452,413.439,402.177,179.372,21.559,152.857
C08657=1098.459,413.686,402.137,179.375,21.567,152.858
C08658=1098.465,413.933,402.098,179.378,21.576,152.860
C08659=1098.470,414.180,402.057,179.379,21.583,152.862
C08660=1098.476,414.427,402.018,179.382,21.592,152.863
C08661=1098.482,414.673,401.978,179.385,21.600,152.865
C08662=1098.488,414.920,401.938,179.387,21.609,152.867
C08663=1098.495,415.166,401.898,179.390,21.617,152.868
C08664=1098.500,415.414,401.858,179.392,21.625,152.870
C08665=1098.506,415.660,401.818,179.395,21.634,152.872
C08666=1098.513,415.907,401.778,179.398,21.642,152.873
C08667=1098.518,416.153,401.739,179.399,21.650,152.875
C08668=1098.524,416.400,401.698,179.402,21.658,152.877
C08669=1098.530,416.647,401.658,179.404,21.667,152.878
C08670=1098.536,416.894,401.619,179.407,21.676,152.880
C08671=1098.542,417.141,401.578,179.409,21.684,152.882
C08672=1098.548,417.387,401.538,179.412,21.693,152.884
C08673=1098.553,417.633,401.497,179.414,21.702,152.886
C08674=1098.560,417.880,401.458,179.417,21.710,152.887
C08675=1098.565,418.127,401.417,179.419,21.719,152.889
C08676=1098.572,418.374,401.377,179.421,21.728,152.891
C08677=1098.578,418.620,401.337,179.424,21.737,152.893
C08678=1098.584,418.867,401.296,179.426,21.745,152.894
C08679=1098.590,419.113,401.256,179.429,21.754,152.896
C08680=1098.596,419.360,401.215,179.431,21.763,152.898
C08681=1098.601,419.606,401.175,179.433,21.772,152.900
C08682=1098.607,419.853,401.135,179.436,21.781,152.902
C08683=1098.613,420.099,401.095,179.438,21.790,152.904
C08684=1098.619,420.346,401.054,179.441,21.798,152.905
C08685=1098.625,420.593,401.014,179.443,21.807,152.907
C08686=1098.631,420.840,400.973,179.445,21.817,152.909
C08687=1098.637,421.086,400.932,179.448,21.826,152.911
C08688=1098.643,421.333,400.892,179.451,21.835,152.913
C08689=1098.649,421.580,400.851,179.453,21.844,152.915
C08690=1098.655,421.826,400.811,179.456,21.853,152.917
C08691=1098.661,422.073,400.770,179.458,21.862,152.919
C08692=1098.667,422.319,400.730,179.460,21.871,152.921
C08693=1098.673,422.566,400.689,179.462,21.880,152.923
C08694=1098.679,422.813,400.648,179.465,21.889,152.924
C08695=1098.685,423.059,400.608,179.467,21.899,152.926
C08696=1098.691,423.305,400.566,179.470,21.909,152.928
C08697=1098.697,423.552,400.526,179.472,21.918,152.930
C08698=1098.702,423.776,400.488,179.474,21.926,152.932
C08699=1098.708,424.001,400.452,179.476,21.935,152.934
C08700=1098.713,424.224,400.415,179.479,21.944,152.936
C08701=1098.718,424.448,400.378,179.480,21.952,152.938
C08702=1098.724,424.673,400.340,179.483,21.961,152.939
C08703=1098.729,424.896,400.303,179.484,21.969,152.941
C08704=1098.735,425.121,400.266,179.487,21.978,152.943
C08705=1098.740,425.345,400.228,179.489,21.987,152.945
C08706=1098.746,425.591,400.187,179.491,21.997,152.947
C08707=1098.752,425.838,400.147,179.494,22.006,152.949
C08708=1098.758,426.084,400.105,179.497,22.016,152.951
C08709=1098.764,426.331,400.065,179.499,22.026,152.953
C08710=1098.770,426.577,400.023,179.501,22.036,152.955
C08711=1098.776,426.825,399.982,179.503,22.045,152.957
C08712=1098.782,427.071,399.941,179.506,22.055,152.960
C08713=1098.789,427.317,399.900,179.508,22.065,152.962
C08714=1098.794,427.563,399.859,179.510,22.075,152.964
C08715=1098.800,427.810,399.817,179.513,22.085,152.966
C08716=1098.806,428.056,399.776,179.515,22.095,152.968
C08717=1098.812,428.303,399.735,179.517,22.105,152.970
C08718=1098.818,428.550,399.693,179.519,22.115,152.972
C08719=1098.824,428.796,399.652,179.522,22.125,152.975
C08720=1098.830,429.042,399.611,179.524,22.135,152.977
C08721=1098.836,429.288,399.569,179.527,22.145,152.979
C08722=1098.842,429.534,399.528,179.528,22.156,152.981
C08723=1098.848,429.781,399.487,179.531,22.165,152.983
C08724=1098.854,430.028,399.445,179.533,22.176,152.986
C08725=1098.860,430.274,399.404,179.535,22.186,152.988
C08726=1098.866,430.521,399.362,179.537,22.196,152.990
C08727=1098.872,430.767,399.321,179.540,22.207,152.992
C08728=1098.878,431.013,399.279,179.542,22.217,152.995
C08729=1098.885,431.260,399.237,179.545,22.228,152.997
C08730=1098.891,431.506,399.196,179.546,22.238,152.999
C08731=1098.897,431.752,399.154,179.549,22.249,153.001
C08732=1098.903,431.998,399.113,179.551,22.260,153.004
C08733=1098.908,432.246,399.071,179.554,22.270,153.006
C08734=1098.915,432.491,399.028,179.556,22.281,153.008
C08735=1098.921,432.737,398.987,179.557,22.291,153.011
C08736=1098.927,432.984,398.946,179.560,22.302,153.013
C08737=1098.933,433.231,398.904,179.562,22.312,153.015
C08738=1098.939,433.477,398.862,179.564,22.323,153.018
C08739=1098.945,433.723,398.819,179.566,22.334,153.020
C08740=1098.950,433.969,398.778,179.569,22.345,153.023
C08741=1098.957,434.216,398.736,179.571,22.356,153.025
C08742=1098.962,434.462,398.694,179.573,22.367,153.028
C08743=1098.968,434.708,398.652,179.576,22.378,153.030
C08744=1098.975,434.955,398.610,179.577,22.389,153.032
C08745=1098.980,435.201,398.568,179.580,22.401,153.035
C08746=1098.986,435.447,398.526,179.582,22.411,153.037
C08747=1098.992,435.693,398.484,179.584,22.423,153.040
C08748=1098.999,435.940,398.441,179.586,22.434,153.042
C08749=1099.005,436.186,398.400,179.588,22.445,153.045
C08750=1099.011,436.431,398.358,179.591,22.457,153.047
C08751=1099.017,436.679,398.315,179.592,22.467,153.050
C08752=1099.023,436.924,398.273,179.595,22.479,153.052
C08753=1099.029,437.172,398.231,179.597,22.490,153.055
C08754=1099.036,437.457,398.182,179.599,22.504,153.058
C08755=1099.043,437.745,398.132,179.602,22.517,153.061
C08756=1099.050,438.033,398.083,179.604,22.531,153.064
C08757=1099.057,438.320,398.033,179.607,22.544,153.067
C08758=1099.063,438.567,397.990,179.608,22.556,153.070
C08759=1099.069,438.812,397.948,179.611,22.567,153.072
C08760=1099.076,439.059,397.906,179.613,22.579,153.075
C08761=1099.082,439.305,397.864,179.615,22.591,153.078
C08762=1099.088,439.552,397.821,179.617,22.602,153.080
C08763=1099.094,439.797,397.778,179.619,22.614,153.083
C08764=1099.101,440.044,397.736,179.622,22.626,153.086
C08765=1099.106,440.290,397.693,179.623,22.638,153.088
C08766=1099.113,440.536,397.650,179.625,22.650,153.091
C08767=1099.119,440.782,397.608,179.628,22.662,153.094
C08768=1099.124,441.028,397.566,179.630,22.675,153.097
C08769=1099.131,441.275,397.523,179.631,22.686,153.099
C08770=1099.136,441.520,397.480,179.634,22.698,153.102
C08771=1099.143,441.766,397.436,179.636,22.711,153.105
C08772=1099.150,442.013,397.394,179.638,22.723,153.108
C08773=1099.155,442.259,397.351,179.640,22.736,153.111
C08774=1099.161,442.505,397.308,179.642,22.748,153.113
C08775=1099.167,442.751,397.266,179.644,22.760,153.116
C08776=1099.174,442.997,397.223,179.646,22.773,153.119
C08777=1099.179,443.243,397.180,179.648,22.785,153.122
C08778=1099.185,443.490,397.137,179.650,22.798,153.125
C08779=1099.192,443.735,397.094,179.652,22.811,153.128
C08780=1099.198,443.981,397.051,179.653,22.822,153.131
C08781=1099.204,444.228,397.008,179.655,22.835,153.134
C08782=1099.209,444.474,396.965,179.656,22.848,153.137
C08783=1099.216,444.720,396.921,179.658,22.861,153.140
C08784=1099.221,444.966,396.878,179.660,22.873,153.143
C08785=1099.228,445.212,396.836,179.660,22.885,153.146
C08786=1099.235,445.496,396.785,179.661,22.900,153.149
C08787=1099.242,445.780,396.735,179.662,22.914,153.153
C08788=1099.250,446.065,396.685,179.663,22.929,153.156
C08789=1099.257,446.349,396.635,179.663,22.943,153.160
C08790=1099.263,446.595,396.592,179.663,22.955,153.163
C08791=1099.269,446.841,396.548,179.663,22.968,153.166
C08792=1099.275,447.087,396.505,179.663,22.980,153.169
C08793=1099.281,447.333,396.462,179.663,22.992,153.172
C08794=1099.287,447.579,396.419,179.663,23.005,153.176
C08795=1099.294,447.825,396.375,179.663,23.018,153.179
C08796=1099.300,448.072,396.332,179.662,23.030,153.182
C08797=1099.305,448.317,396.288,179.661,23.042,153.185
C08798=1099.312,448.564,396.245,179.660,23.054,153.188
C08799=1099.318,448.810,396.201,179.659,23.066,153.192
C08800=1099.323,449.057,396.158,179.658,23.079,153.195
C08801=1099.329,449.302,396.114,179.658,23.091,153.198
C08802=1099.336,449.548,396.070,179.657,23.104,153.202
C08803=1099.342,449.794,396.027,179.655,23.115,153.205
C08804=1099.348,450.040,395.984,179.654,23.128,153.208
C08805=1099.355,450.286,395.940,179.652,23.140,153.211
C08806=1098.959,450.277,395.789,179.589,23.358,153.276
C08807=1098.952,450.032,395.832,179.590,23.347,153.273
C08808=1098.946,449.786,395.876,179.592,23.335,153.269
C08809=1098.940,449.540,395.919,179.593,23.322,153.266
C08810=1098.933,449.294,395.963,179.594,23.309,153.263
C08811=1098.927,449.048,396.006,179.595,23.298,153.259
C08812=1098.921,448.802,396.050,179.596,23.285,153.256
C08813=1098.915,448.557,396.093,179.597,23.273,153.253
C08814=1098.909,448.310,396.137,179.598,23.260,153.250
C08815=1098.903,448.064,396.180,179.598,23.248,153.246
C08816=1098.896,447.818,396.224,179.598,23.235,153.243
C08817=1098.890,447.571,396.267,179.599,23.223,153.240
C08818=1098.884,447.326,396.311,179.599,23.211,153.237
C08819=1098.878,447.080,396.354,179.599,23.198,153.234
C08820=1098.872,446.834,396.398,179.600,23.186,153.230
C08821=1098.866,446.587,396.441,179.600,23.173,153.227
C08822=1098.860,446.342,396.485,179.598,23.160,153.224
C08823=1098.854,446.095,396.528,179.598,23.148,153.221
C08824=1098.847,445.849,396.571,179.598,23.135,153.218
C08825=1098.842,445.603,396.614,179.597,23.123,153.215
C08826=1098.835,445.357,396.658,179.597,23.111,153.212
C08827=1098.829,445.111,396.701,179.595,23.098,153.209
C08828=1098.823,444.865,396.745,179.594,23.085,153.206
C08829=1098.817,444.619,396.788,179.593,23.073,153.203
C08830=1098.810,444.373,396.831,179.592,23.060,153.200
C08831=1098.804,444.127,396.874,179.590,23.047,153.197
C08832=1098.798,443.881,396.917,179.588,23.035,153.194
C08833=1098.792,443.634,396.960,179.586,23.022,153.191
C08834=1098.786,443.389,397.004,179.584,23.009,153.188
C08835=1098.780,443.142,397.047,179.582,22.997,153.185
C08836=1098.773,442.896,397.089,179.580,22.984,153.182
C08837=1098.768,442.651,397.133,179.578,22.971,153.179
C08838=1098.762,442.404,397.176,179.575,22.959,153.176
C08839=1098.756,442.158,397.219,179.574,22.947,153.174
C08840=1098.749,441.912,397.261,179.572,22.934,153.171
C08841=1098.744,441.666,397.304,179.569,22.922,153.168
C08842=1098.738,441.419,397.347,179.567,22.910,153.165
C08843=1098.731,441.174,397.389,179.565,22.897,153.162
C08844=1098.725,440.927,397.432,179.563,22.886,153.160
C08845=1098.720,440.681,397.475,179.561,22.873,153.157
C08846=1098.713,440.435,397.518,179.559,22.861,153.154
C08847=1098.707,440.188,397.561,179.556,22.849,153.151
C08848=1098.700,439.943,397.603,179.555,22.838,153.149
C08849=1098.694,439.696,397.646,179.552,22.825,153.146
C08850=1098.688,439.451,397.688,179.550,22.813,153.143
C08851=1098.682,439.204,397.732,179.548,22.801,153.141
C08852=1098.676,438.959,397.774,179.546,22.790,153.138
C08853=1098.670,438.712,397.817,179.544,22.778,153.135
C08854=1098.664,438.466,397.858,179.541,22.766,153.133
C08855=1098.655,438.148,397.914,179.539,22.751,153.129
C08856=1098.648,437.831,397.968,179.536,22.736,153.126
C08857=1098.640,437.513,398.022,179.533,22.722,153.123
C08858=1098.632,437.196,398.078,179.530,22.706,153.119
C08859=1098.626,436.950,398.119,179.528,22.695,153.117
C08860=1098.620,436.703,398.162,179.526,22.684,153.114
C08861=1098.614,436.458,398.204,179.523,22.672,153.112
C08862=1098.608,436.212,398.246,179.522,22.661,153.109
C08863=1098.602,435.965,398.289,179.519,22.650,153.107
C08864=1098.596,435.719,398.330,179.517,22.638,153.104
C08865=1098.590,435.472,398.374,179.515,22.627,153.102
C08866=1098.584,435.226,398.415,179.512,22.616,153.099
C08867=1098.577,434.980,398.457,179.511,22.605,153.097
C08868=1098.572,434.733,398.500,179.508,22.594,153.094
C08869=1098.565,434.488,398.542,179.506,22.583,153.092
C08870=1098.559,434.241,398.583,179.504,22.571,153.089
C08871=1098.554,433.994,398.626,179.501,22.560,153.087
C08872=1098.547,433.749,398.668,179.499,22.550,153.084
C08873=1098.541,433.502,398.709,179.497,22.538,153.082
C08874=1098.536,433.256,398.751,179.495,22.528,153.079
C08875=1098.530,433.009,398.793,179.492,22.517,153.077
C08876=1098.523,432.763,398.835,179.490,22.506,153.075
C08877=1098.517,432.517,398.877,179.487,22.495,153.072
C08878=1098.511,432.270,398.919,179.485,22.485,153.070
C08879=1098.505,432.024,398.960,179.483,22.474,153.068
C08880=1098.500,431.778,399.002,179.481,22.463,153.065
C08881=1098.493,431.532,399.044,179.479,22.453,153.063
C08882=1098.487,431.285,399.086,179.476,22.442,153.061
C08883=1098.481,431.039,399.128,179.474,22.432,153.058
C08884=1098.475,430.793,399.169,179.472,22.421,153.056
C08885=1098.469,430.546,399.211,179.470,22.411,153.054
C08886=1098.462,430.300,399.252,179.467,22.401,153.052
C08887=1098.456,430.053,399.294,179.465,22.390,153.049
C08888=1098.451,429.807,399.335,179.463,22.380,153.047
C08889=1098.445,429.561,399.377,179.460,22.369,153.045
C08890=1098.439,429.315,399.418,179.458,22.359,153.043
C08891=1098.433,429.068,399.459,179.456,22.349,153.040
C08892=1098.426,428.821,399.501,179.453,22.339,153.038
C08893=1098.421,428.575,399.542,179.451,22.329,153.036
C08894=1098.415,428.329,399.584,179.449,22.319,153.034
C08895=1098.409,428.082,399.625,179.446,22.308,153.032
C08896=1098.402,427.835,399.667,179.444,22.298,153.030
C08897=1098.396,427.589,399.708,179.442,22.288,153.027
C08898=1098.390,427.342,399.749,179.439,22.279,153.025
C08899=1098.385,427.096,399.791,179.437,22.269,153.023
C08900=1098.379,426.849,399.831,179.434,22.259,153.021
C08901=1098.372,426.604,399.872,179.432,22.248,153.019
C08902=1098.366,426.357,399.914,179.429,22.239,153.017
C08903=1098.360,426.110,399.955,179.427,22.229,153.015
C08904=1098.354,425.864,399.996,179.425,22.220,153.013
C08905=1098.348,425.617,400.037,179.422,22.209,153.011
C08906=1098.342,425.371,400.078,179.420,22.200,153.009
C08907=1098.337,425.146,400.116,179.418,22.191,153.007
C08908=1098.332,424.922,400.153,179.416,22.182,153.005
C08909=1098.326,424.698,400.191,179.413,22.173,153.003
C08910=1098.320,424.473,400.228,179.412,22.165,153.001
C08911=1098.315,424.249,400.265,179.409,22.156,152.999
C08912=1098.310,424.024,400.302,179.407,22.147,152.997
C08913=1098.304,423.800,400.340,179.405,22.139,152.996
C08914=1098.299,423.575,400.376,179.402,22.130,152.994
C08915=1098.293,423.328,400.417,179.400,22.121,152.992
C08916=1098.287,423.083,400.458,179.398,22.111,152.990
C08917=1098.281,422.836,400.499,179.396,22.102,152.988
C08918=1098.275,422.589,400.539,179.393,22.092,152.986
C08919=1098.269,422.343,400.580,179.390,22.083,152.984
C08920=1098.263,422.096,400.621,179.388,22.074,152.982
C08921=1098.258,421.849,400.662,179.386,22.065,152.980
C08922=1098.251,421.603,400.702,179.383,22.056,152.978
C08923=1098.245,421.355,400.743,179.381,22.047,152.976
C08924=1098.238,421.109,400.784,179.378,22.038,152.974
C08925=1098.233,420.863,400.824,179.376,22.028,152.973
C08926=1098.227,420.617,400.864,179.374,22.019,152.971
C08927=1098.221,420.370,400.905,179.371,22.010,152.969
C08928=1098.215,420.123,400.945,179.369,22.001,152.967
C08929=1098.209,419.877,400.986,179.366,21.992,152.965
C08930=1098.203,419.630,401.026,179.363,21.983,152.963
C08931=1098.196,419.362,401.070,179.361,21.974,152.961
C08932=1098.189,419.094,401.115,179.358,21.964,152.959
C08933=1098.183,418.826,401.158,179.356,21.954,152.957
C08934=1098.177,418.558,401.202,179.353,21.944,152.955
C08935=1098.171,418.312,401.242,179.350,21.936,152.953
C08936=1098.165,418.065,401.283,179.347,21.927,152.952
C08937=1098.159,417.819,401.323,179.345,21.918,152.950
C08938=1098.153,417.572,401.363,179.343,21.909,152.948
C08939=1098.147,417.326,401.404,179.340,21.901,152.946
C08940=1098.141,417.079,401.444,179.338,21.892,152.945
C08941=1098.135,416.832,401.484,179.336,21.884,152.943
C08942=1098.130,416.585,401.525,179.333,21.875,152.941
C08943=1098.124,416.339,401.564,179.331,21.867,152.939
C08944=1098.118,416.092,401.604,179.328,21.858,152.938
C08945=1098.111,415.845,401.644,179.326,21.849,152.936
C08946=1098.106,415.599,401.685,179.323,21.841,152.934
C08947=1098.099,415.352,401.725,179.320,21.832,152.932
C08948=1098.093,415.105,401.764,179.318,21.824,152.931
C08949=1098.087,414.858,401.804,179.315,21.816,152.929
C08950=1098.082,414.611,401.844,179.313,21.807,152.927
C08951=1098.076,414.365,401.884,179.311,21.799,152.926
C08952=1098.070,414.119,401.924,179.308,21.791,152.924
C08953=1098.063,413.871,401.964,179.306,21.782,152.922
C08954=1098.057,413.625,402.004,179.303,21.774,152.921
C08955=1098.052,413.377,402.044,179.300,21.766,152.919
C08956=1098.046,413.132,402.084,179.297,21.758,152.918
C08957=1098.040,412.885,402.123,179.296,21.750,152.916
C08958=1098.034,412.637,402.163,179.293,21.742,152.914
C08959=1098.027,412.391,402.203,179.290,21.733,152.913
C08960=1098.022,412.144,402.242,179.287,21.725,152.911
C08961=1098.016,411.898,402.283,179.286,21.717,152.909
C08962=1098.010,411.650,402.322,179.283,21.709,152.908
C08963=1098.000,411.237,402.388,179.278,21.695,152.905
C08964=1097.990,410.824,402.454,179.274,21.682,152.903
C08965=1097.980,410.410,402.521,179.270,21.669,152.900
C08966=1097.970,409.996,402.588,179.265,21.656,152.897
C08967=1097.965,409.749,402.627,179.263,21.648,152.896
C08968=1097.959,409.502,402.666,179.261,21.640,152.894
C08969=1097.953,409.255,402.706,179.258,21.632,152.893
C08970=1097.947,409.009,402.745,179.256,21.625,152.891
C08971=1097.941,408.762,402.784,179.253,21.617,152.890
C08972=1097.935,408.514,402.823,179.250,21.609,152.888
C08973=1097.929,408.269,402.863,179.248,21.602,152.887
C08974=1097.923,408.021,402.903,179.246,21.594,152.885
C08975=1097.918,407.775,402.942,179.243,21.586,152.884
C08976=1097.912,407.528,402.981,179.241,21.579,152.882
C08977=1097.906,407.281,403.021,179.238,21.571,152.881
C08978=1097.900,407.034,403.060,179.235,21.563,152.879
C08979=1097.894,406.787,403.099,179.233,21.556,152.878
C08980=1097.889,406.540,403.137,179.230,21.548,152.876
C08981=1097.883,406.293,403.177,179.228,21.541,152.875
C08982=1097.876,406.046,403.216,179.225,21.533,152.873
C08983=1097.871,405.800,403.255,179.222,21.525,152.872
C08984=1097.865,405.553,403.294,179.220,21.518,152.871
C08985=1097.859,405.306,403.333,179.217,21.510,152.869
C08986=1097.853,405.059,403.373,179.215,21.504,152.868
C08987=1097.848,404.813,403.412,179.212,21.496,152.866
C08988=1097.841,404.565,403.450,179.210,21.489,152.865
C08989=1097.836,404.319,403.489,179.207,21.481,152.864
C08990=1097.829,404.072,403.528,179.205,21.475,152.862
C08991=1097.823,403.824,403.568,179.202,21.467,152.861
C08992=1097.817,403.578,403.606,179.200,21.460,152.859
C08993=1097.811,403.331,403.645,179.197,21.452,152.858
C08994=1097.806,403.084,403.684,179.194,21.445,152.857
C08995=1097.799,402.837,403.722,179.191,21.438,152.855
C08996=1097.794,402.590,403.761,179.189,21.431,152.854
C08997=1097.788,402.343,403.801,179.186,21.424,152.853
C08998=1097.782,402.096,403.838,179.184,21.417,152.851
C08999=1097.776,401.849,403.878,179.181,21.409,152.850
C09000=1097.771,401.602,403.916,179.179,21.403,152.849
C09001=1097.765,401.356,403.955,179.176,21.395,152.847
C09002=1097.759,401.108,403.993,179.174,21.389,152.846
C09003=1097.753,400.862,404.032,179.170,21.382,152.845
C09004=1097.747,400.614,404.071,179.168,21.375,152.844
C09005=1097.741,400.368,404.110,179.166,21.368,152.842
C09006=1097.735,400.121,404.147,179.163,21.361,152.841
C09007=1097.729,399.874,404.187,179.161,21.354,152.840
C09008=1097.723,399.627,404.225,179.157,21.347,152.838
C09009=1097.718,399.380,404.263,179.155,21.340,152.837
C09010=1097.711,399.133,404.302,179.153,21.333,152.836
C09011=1097.706,398.886,404.340,179.150,21.326,152.835
C09012=1097.700,398.639,404.378,179.147,21.320,152.833
C09013=1097.694,398.393,404.417,179.144,21.312,152.832
C09014=1097.688,398.145,404.455,179.142,21.306,152.831
C09015=1097.683,397.928,404.489,179.139,21.300,152.830
C09016=1097.678,397.711,404.523,179.138,21.294,152.829
C09017=1097.673,397.493,404.557,179.135,21.288,152.828
C09018=1097.668,397.276,404.591,179.133,21.282,152.827
C09019=1097.662,397.059,404.624,179.131,21.277,152.825
C09020=1097.657,396.842,404.657,179.128,21.271,152.825
C09021=1097.652,396.624,404.691,179.125,21.265,152.823
C09022=1097.647,396.407,404.725,179.124,21.259,152.822
C09023=1097.641,396.160,404.763,179.121,21.252,152.821
C09024=1097.635,395.913,404.802,179.118,21.246,152.820
C09025=1097.630,395.666,404.839,179.116,21.239,152.819
C09026=1097.623,395.419,404.877,179.113,21.233,152.818
C09027=1097.618,395.172,404.916,179.110,21.226,152.816
C09028=1097.612,394.925,404.954,179.108,21.220,152.815
C09029=1097.606,394.678,404.991,179.105,21.214,152.814
C09030=1097.599,394.431,405.030,179.102,21.207,152.813
C09031=1097.594,394.184,405.068,179.100,21.201,152.812
C09032=1097.588,393.938,405.106,179.097,21.195,152.811
C09033=1097.582,393.691,405.144,179.094,21.187,152.810
C09034=1097.576,393.443,405.182,179.091,21.181,152.809
C09035=1097.571,393.196,405.220,179.089,21.175,152.807
C09036=1097.565,392.949,405.257,179.086,21.169,152.806
C09037=1097.559,392.702,405.295,179.083,21.162,152.805
C09038=1097.553,392.455,405.333,179.081,21.156,152.804
C09039=1097.547,392.208,405.371,179.078,21.150,152.803
C09040=1097.542,391.961,405.409,179.076,21.144,152.802
C09041=1097.536,391.714,405.447,179.073,21.137,152.801
C09042=1097.530,391.467,405.485,179.070,21.131,152.800
C09043=1097.524,391.220,405.522,179.067,21.125,152.799
C09044=1097.518,390.973,405.560,179.064,21.119,152.798
C09045=1097.512,390.726,405.598,179.062,21.113,152.797
C09046=1097.506,390.479,405.636,179.059,21.106,152.796
C09047=1097.500,390.232,405.673,179.056,21.100,152.794
C09048=1097.494,389.985,405.710,179.054,21.094,152.793
C09049=1097.488,389.738,405.748,179.051,21.089,152.792
C09050=1097.483,389.492,405.786,179.048,21.082,152.791
C09051=1097.476,389.243,405.823,179.045,21.076,152.790
C09052=1097.470,388.997,405.861,179.042,21.070,152.789
C09053=1097.465,388.750,405.899,179.040,21.064,152.788
C09054=1097.459,388.503,405.936,179.037,21.058,152.787
C09055=1097.453,388.256,405.974,179.034,21.052,152.786
C09056=1097.447,388.009,406.011,179.032,21.046,152.785
C09057=1097.441,387.762,406.048,179.028,21.040,152.784
C09058=1097.435,387.515,406.086,179.026,21.034,152.783
C09059=1097.429,387.268,406.123,179.023,21.028,152.782
C09060=1097.423,387.021,406.160,179.020,21.023,152.781
C09061=1097.418,386.774,406.197,179.018,21.017,152.780
C09062=1097.412,386.527,406.235,179.015,21.011,152.779
C09063=1097.406,386.280,406.272,179.012,21.005,152.778
C09064=1097.400,386.033,406.310,179.009,20.999,152.777
C09065=1097.395,385.786,406.347,179.006,20.993,152.776
C09066=1097.389,385.538,406.384,179.004,20.987,152.775
C09067=1097.383,385.292,406.421,179.001,20.982,152.775
C09068=1097.377,385.045,406.458,178.998,20.976,152.774
C09069=1097.371,384.798,406.496,178.996,20.970,152.773
C09070=1097.365,384.550,406.533,178.993,20.964,152.772
C09071=1097.360,384.339,406.565,178.990,20.959,152.771
C09072=1097.356,384.128,406.596,178.988,20.954,152.770
C09073=1097.351,383.917,406.628,178.986,20.949,152.769
C09074=1097.346,383.706,406.660,178.983,20.944,152.768
C09075=1097.341,383.495,406.692,178.981,20.939,152.768
C09076=1097.336,383.285,406.723,178.979,20.935,152.767
C09077=1097.331,383.073,406.755,178.976,20.930,152.766
C09078=1097.327,382.863,406.786,178.974,20.925,152.765
C09079=1097.321,382.616,406.823,178.971,20.920,152.764
C09080=1097.315,382.368,406.860,178.968,20.914,152.763
C09081=1097.309,382.122,406.897,178.965,20.909,152.763
C09082=1097.303,381.875,406.934,178.963,20.903,152.762
C09083=1097.297,381.627,406.971,178.960,20.897,152.761
C09084=1097.291,381.380,407.007,178.957,20.892,152.760
C09085=1097.285,381.133,407.044,178.954,20.886,152.759
C09086=1097.280,380.885,407.081,178.951,20.881,152.758
C09087=1097.273,380.638,407.118,178.949,20.875,152.757
C09088=1097.268,380.391,407.155,178.946,20.870,152.757
C09089=1097.261,380.144,407.191,178.943,20.865,152.756
C09090=1097.256,379.897,407.228,178.940,20.859,152.755
C09091=1097.251,379.650,407.265,178.937,20.854,152.754
C09092=1097.244,379.403,407.302,178.934,20.848,152.753
C09093=1097.239,379.156,407.339,178.932,20.843,152.752
C09094=1097.233,378.909,407.375,178.929,20.838,152.751
C09095=1097.227,378.661,407.412,178.926,20.833,152.751
C09096=1097.221,378.414,407.449,178.923,20.827,152.750
C09097=1097.215,378.167,407.486,178.920,20.822,152.749
C09098=1097.209,377.920,407.522,178.917,20.816,152.748
C09099=1097.204,377.672,407.558,178.914,20.811,152.747
C09100=1097.198,377.425,407.594,178.911,20.806,152.747
C09101=1097.192,377.178,407.631,178.909,20.800,152.746
C09102=1097.186,376.932,407.668,178.906,20.795,152.745
C09103=1097.181,376.684,407.705,178.903,20.790,152.744
C09104=1097.175,376.437,407.740,178.900,20.784,152.743
C09105=1097.169,376.189,407.777,178.897,20.779,152.742
C09106=1097.163,375.942,407.814,178.894,20.774,152.742
